C01785=1051.744,309.369,-107.707,172.758,38.228,157.251
C01786=1051.737,309.122,-107.673,172.754,38.225,157.251
C01787=1051.730,308.873,-107.640,172.750,38.221,157.250
C01788=1051.724,308.627,-107.607,172.747,38.218,157.249
C01789=1051.717,308.378,-107.574,172.743,38.214,157.248
C01790=1051.710,308.131,-107.541,172.739,38.211,157.247
C01791=1051.703,307.883,-107.507,172.737,38.207,157.246
C01792=1051.697,307.635,-107.474,172.733,38.203,157.245
C01793=1051.691,307.388,-107.441,172.729,38.200,157.245
C01794=1051.683,307.140,-107.409,172.725,38.197,157.244
C01795=1051.676,306.893,-107.375,172.722,38.193,157.243
C01796=1051.669,306.644,-107.342,172.719,38.189,157.242
C01797=1051.663,306.397,-107.310,172.715,38.186,157.241
C01798=1051.657,306.149,-107.277,172.712,38.183,157.240
C01799=1051.650,305.902,-107.243,172.708,38.179,157.239
C01800=1051.643,305.654,-107.210,172.704,38.175,157.239
C01801=1051.637,305.406,-107.178,172.701,38.172,157.238
C01802=1051.629,305.158,-107.145,172.698,38.168,157.237
C01803=1051.623,304.877,-107.108,172.694,38.164,157.236
C01804=1051.615,304.595,-107.070,172.690,38.160,157.235
C01805=1051.607,304.314,-107.033,172.685,38.156,157.234
C01806=1051.600,304.032,-106.996,172.682,38.152,157.233
C01807=1051.593,303.784,-106.963,172.679,38.149,157.232
C01808=1051.586,303.536,-106.930,172.675,38.145,157.231
C01809=1051.580,303.289,-106.898,172.671,38.141,157.230
C01810=1051.574,303.041,-106.865,172.668,38.138,157.230
C01811=1051.567,302.793,-106.832,172.665,38.135,157.229
C01812=1051.561,302.545,-106.799,172.661,38.131,157.228
C01813=1051.554,302.298,-106.766,172.658,38.128,157.227
C01814=1051.547,302.050,-106.734,172.655,38.124,157.226
C01815=1051.541,301.803,-106.701,172.651,38.120,157.225
C01816=1051.534,301.555,-106.668,172.648,38.117,157.225
C01817=1051.528,301.307,-106.636,172.644,38.114,157.224
C01818=1051.521,301.059,-106.603,172.641,38.110,157.223
C01819=1051.515,300.812,-106.570,172.638,38.106,157.222
C01820=1051.508,300.565,-106.538,172.634,38.103,157.221
C01821=1051.501,300.316,-106.505,172.631,38.099,157.220
C01822=1051.495,300.069,-106.472,172.628,38.096,157.220
C01823=1051.489,299.820,-106.440,172.624,38.093,157.219
C01824=1051.483,299.573,-106.407,172.621,38.089,157.218
C01825=1051.476,299.326,-106.375,172.618,38.085,157.217
C01826=1051.469,299.078,-106.342,172.614,38.082,157.216
C01827=1051.463,298.830,-106.310,172.611,38.078,157.215
C01828=1051.457,298.582,-106.278,172.608,38.075,157.215
C01829=1051.450,298.334,-106.245,172.604,38.072,157.214
C01830=1051.443,298.087,-106.212,172.601,38.068,157.213
C01831=1051.437,297.838,-106.180,172.598,38.065,157.212
C01832=1051.431,297.591,-106.148,172.595,38.061,157.211
C01833=1051.425,297.343,-106.115,172.591,38.057,157.210
C01834=1051.419,297.095,-106.083,172.587,38.054,157.210
C01835=1051.412,296.848,-106.051,172.585,38.051,157.209
C01836=1051.405,296.600,-106.018,172.581,38.047,157.208
C01837=1051.399,296.352,-105.986,172.578,38.044,157.207
C01838=1051.392,296.105,-105.954,172.575,38.040,157.206
C01839=1051.386,295.856,-105.922,172.571,38.037,157.205
C01840=1051.379,295.609,-105.890,172.569,38.033,157.205
C01841=1051.373,295.361,-105.858,172.565,38.030,157.204
C01842=1051.366,295.114,-105.825,172.561,38.027,157.203
C01843=1051.360,294.865,-105.793,172.559,38.023,157.202
C01844=1051.353,294.617,-105.761,172.555,38.020,157.201
C01845=1051.347,294.369,-105.729,172.552,38.016,157.201
C01846=1051.340,294.122,-105.697,172.549,38.013,157.200
C01847=1051.334,293.874,-105.665,172.545,38.010,157.199
C01848=1051.327,293.626,-105.633,172.542,38.006,157.198
C01849=1051.320,293.379,-105.601,172.539,38.003,157.197
C01850=1051.314,293.130,-105.569,172.536,37.999,157.197
C01851=1051.307,292.882,-105.538,172.533,37.996,157.196
C01852=1051.300,292.635,-105.506,172.529,37.993,157.195
C01853=1051.294,292.387,-105.474,172.526,37.990,157.194
C01854=1051.287,292.139,-105.442,172.523,37.986,157.193
C01855=1051.281,291.891,-105.410,172.520,37.983,157.193
C01856=1051.274,291.644,-105.378,172.516,37.979,157.192
C01857=1051.268,291.396,-105.346,172.513,37.976,157.191
C01858=1051.262,291.147,-105.314,172.510,37.972,157.190
C01859=1051.255,290.882,-105.280,172.506,37.969,157.189
C01860=1051.247,290.617,-105.247,172.503,37.966,157.189
C01861=1051.240,290.351,-105.213,172.500,37.962,157.188
C01862=1051.233,290.085,-105.179,172.496,37.958,157.187
C01863=1051.226,289.838,-105.147,172.493,37.955,157.186
C01864=1051.220,289.589,-105.115,172.490,37.952,157.185
C01865=1051.213,289.341,-105.083,172.487,37.949,157.185
C01866=1051.207,289.094,-105.052,172.484,37.945,157.184
C01867=1051.201,288.846,-105.020,172.480,37.942,157.183
C01868=1051.195,288.598,-104.989,172.478,37.938,157.182
C01869=1051.188,288.350,-104.957,172.474,37.935,157.181
C01870=1051.181,288.102,-104.926,172.471,37.932,157.181
C01871=1051.175,287.854,-104.894,172.468,37.929,157.180
C01872=1051.168,287.606,-104.862,172.465,37.925,157.179
C01873=1051.162,287.358,-104.831,172.462,37.922,157.178
C01874=1051.155,287.110,-104.800,172.459,37.919,157.178
C01875=1051.148,286.863,-104.768,172.455,37.915,157.177
C01876=1051.142,286.615,-104.737,172.453,37.912,157.176
C01877=1051.135,286.367,-104.706,172.449,37.909,157.175
C01878=1051.129,286.120,-104.674,172.447,37.906,157.175
C01879=1051.122,285.871,-104.644,172.443,37.902,157.174
C01880=1051.116,285.623,-104.612,172.440,37.899,157.173
C01881=1051.109,285.375,-104.581,172.437,37.896,157.172
C01882=1051.102,285.127,-104.549,172.434,37.892,157.171
C01883=1051.095,284.879,-104.518,172.431,37.889,157.171
C01884=1051.089,284.632,-104.486,172.428,37.886,157.170
C01885=1051.083,284.384,-104.456,172.424,37.883,157.169
C01886=1051.076,284.136,-104.425,172.422,37.879,157.168
C01887=1051.069,283.888,-104.393,172.418,37.876,157.168
C01888=1051.063,283.640,-104.361,172.416,37.873,157.167
C01889=1051.057,283.391,-104.330,172.412,37.870,157.166
C01890=1051.051,283.144,-104.299,172.409,37.866,157.165
C01891=1051.044,282.896,-104.268,172.406,37.863,157.165
C01892=1051.038,282.648,-104.237,172.403,37.860,157.164
C01893=1051.031,282.400,-104.206,172.401,37.856,157.163
C01894=1051.024,282.152,-104.174,172.397,37.853,157.162
C01895=1051.018,281.904,-104.144,172.394,37.850,157.162
C01896=1051.012,281.656,-104.113,172.391,37.847,157.161
C01897=1051.005,281.408,-104.081,172.388,37.844,157.160
C01898=1050.999,281.160,-104.050,172.385,37.840,157.159
C01899=1050.992,280.912,-104.019,172.382,37.837,157.159
C01900=1050.986,280.664,-103.989,172.379,37.833,157.158
C01901=1050.979,280.416,-103.957,172.376,37.830,157.157
C01902=1050.973,280.169,-103.926,172.373,37.827,157.156
C01903=1050.967,279.920,-103.895,172.370,37.824,157.155
C01904=1050.960,279.672,-103.864,172.367,37.821,157.155
C01905=1050.954,279.424,-103.834,172.365,37.817,157.154
C01906=1050.947,279.177,-103.803,172.361,37.814,157.153
C01907=1050.940,278.928,-103.772,172.358,37.811,157.153
C01908=1050.934,278.680,-103.741,172.355,37.807,157.152
C01909=1050.928,278.433,-103.710,172.352,37.805,157.151
C01910=1050.921,278.184,-103.680,172.349,37.801,157.150
C01911=1050.914,277.937,-103.649,172.346,37.798,157.150
C01912=1050.908,277.689,-103.618,172.344,37.795,157.149
C01913=1050.902,277.440,-103.588,172.340,37.791,157.148
C01914=1050.895,277.192,-103.556,172.337,37.788,157.147
C01915=1050.889,276.938,-103.525,172.335,37.785,157.147
C01916=1050.882,276.684,-103.493,172.331,37.782,157.146
C01917=1050.875,276.430,-103.462,172.329,37.779,157.145
C01918=1050.868,276.175,-103.431,172.325,37.775,157.144
C01919=1050.862,275.927,-103.400,172.322,37.772,157.144
C01920=1050.855,275.679,-103.370,172.320,37.769,157.143
C01921=1050.849,275.432,-103.339,172.316,37.765,157.142
C01922=1050.843,275.184,-103.308,172.314,37.762,157.141
C01923=1050.836,274.935,-103.278,172.310,37.759,157.141
C01924=1050.830,274.688,-103.248,172.308,37.756,157.140
C01925=1050.823,274.439,-103.217,172.305,37.753,157.139
C01926=1050.816,274.191,-103.186,172.302,37.750,157.138
C01927=1050.810,273.944,-103.156,172.299,37.746,157.138
C01928=1050.803,273.695,-103.125,172.296,37.743,157.137
C01929=1050.798,273.447,-103.095,172.293,37.740,157.136
C01930=1050.791,273.199,-103.065,172.290,37.737,157.135
C01931=1050.785,272.951,-103.034,172.288,37.734,157.135
C01932=1050.778,272.703,-103.004,172.284,37.730,157.134
C01933=1050.771,272.454,-102.974,172.282,37.727,157.133
C01934=1050.765,272.207,-102.943,172.279,37.724,157.133
C01935=1050.759,271.959,-102.912,172.276,37.721,157.132
C01936=1050.752,271.711,-102.882,172.273,37.717,157.131
C01937=1050.746,271.463,-102.851,172.270,37.715,157.130
C01938=1050.739,271.215,-102.822,172.268,37.711,157.130
C01939=1050.733,270.967,-102.791,172.264,37.708,157.129
C01940=1050.726,270.719,-102.762,172.262,37.705,157.128
C01941=1050.720,270.470,-102.731,172.259,37.702,157.128
C01942=1050.713,270.222,-102.701,172.256,37.698,157.127
C01943=1050.707,269.974,-102.671,172.253,37.695,157.126
C01944=1050.700,269.726,-102.640,172.250,37.692,157.125
C01945=1050.694,269.478,-102.610,172.248,37.689,157.125
C01946=1050.687,269.230,-102.580,172.244,37.686,157.124
C01947=1050.681,268.982,-102.550,172.242,37.683,157.123
C01948=1050.674,268.734,-102.520,172.239,37.680,157.123
C01949=1050.668,268.486,-102.489,172.237,37.676,157.122
C01950=1050.662,268.238,-102.460,172.233,37.673,157.121
C01951=1050.655,267.989,-102.429,172.231,37.670,157.120
C01952=1050.649,267.742,-102.400,172.228,37.667,157.120
C01953=1050.642,267.493,-102.370,172.225,37.664,157.119
C01954=1050.636,267.245,-102.340,172.222,37.661,157.118
C01955=1050.629,266.997,-102.310,172.220,37.658,157.117
C01956=1050.622,266.749,-102.280,172.217,37.654,157.117
C01957=1050.616,266.501,-102.249,172.213,37.651,157.116
C01958=1050.610,266.253,-102.220,172.211,37.648,157.115
C01959=1050.603,266.004,-102.190,172.208,37.645,157.115
C01960=1050.597,265.757,-102.160,172.206,37.642,157.114
C01961=1050.590,265.508,-102.130,172.203,37.639,157.113
C01962=1050.584,265.260,-102.100,172.200,37.636,157.112
C01963=1050.578,265.012,-102.070,172.197,37.632,157.112
C01964=1050.571,264.764,-102.041,172.195,37.629,157.111
C01965=1050.565,264.516,-102.011,172.192,37.626,157.110
C01966=1050.558,264.268,-101.980,172.189,37.623,157.110
C01967=1050.552,264.019,-101.951,172.186,37.619,157.109
C01968=1050.546,263.772,-101.921,172.183,37.617,157.108
C01969=1050.539,263.523,-101.892,172.181,37.614,157.108
C01970=1050.532,263.275,-101.862,172.178,37.610,157.107
C01971=1050.526,263.025,-101.832,172.175,37.607,157.106
C01972=1050.520,262.776,-101.802,172.172,37.604,157.105
C01973=1050.513,262.526,-101.772,172.170,37.601,157.105
C01974=1050.507,262.275,-101.742,172.167,37.598,157.104
C01975=1050.500,262.026,-101.713,172.165,37.594,157.103
C01976=1050.493,261.779,-101.683,172.161,37.592,157.103
C01977=1050.487,261.531,-101.654,172.159,37.589,157.102
C01978=1050.479,261.283,-101.624,172.156,37.586,157.101
C01979=1050.473,261.035,-101.595,172.154,37.582,157.100
C01980=1050.466,260.786,-101.566,172.150,37.579,157.100
C01981=1050.459,260.538,-101.536,172.148,37.576,157.099
C01982=1050.453,260.290,-101.507,172.145,37.573,157.098
C01983=1050.446,260.041,-101.478,172.143,37.570,157.098
C01984=1050.440,259.794,-101.448,172.140,37.567,157.097
C01985=1050.434,259.546,-101.419,172.138,37.564,157.096
C01986=1050.427,259.297,-101.390,172.134,37.561,157.096
C01987=1050.420,259.049,-101.361,172.132,37.558,157.095
C01988=1050.414,258.801,-101.331,172.129,37.555,157.094
C01989=1050.407,258.553,-101.301,172.127,37.552,157.094
C01990=1050.401,258.304,-101.272,172.124,37.548,157.093
C01991=1050.395,258.056,-101.243,172.122,37.546,157.092
C01992=1050.387,257.808,-101.213,172.118,37.543,157.092
C01993=1050.381,257.560,-101.184,172.115,37.539,157.091
C01994=1050.375,257.312,-101.155,172.113,37.536,157.090
C01995=1050.368,257.063,-101.126,172.111,37.533,157.089
C01996=1050.362,256.815,-101.097,172.108,37.530,157.089
C01997=1050.356,256.567,-101.068,172.105,37.527,157.088
C01998=1050.349,256.319,-101.038,172.103,37.524,157.087
C01999=1050.342,256.070,-101.008,172.099,37.521,157.087
C02000=1050.336,255.822,-100.979,172.097,37.518,157.086
C02001=1050.329,255.574,-100.951,172.094,37.515,157.085
C02002=1050.323,255.326,-100.922,172.092,37.512,157.085
C02003=1050.316,255.077,-100.893,172.089,37.508,157.084
C02004=1050.310,254.829,-100.864,172.087,37.505,157.083
C02005=1050.303,254.581,-100.834,172.084,37.502,157.083
C02006=1050.297,254.333,-100.805,172.082,37.499,157.082
C02007=1050.291,254.085,-100.776,172.079,37.496,157.081
C02008=1050.284,253.836,-100.747,172.077,37.493,157.080
C02009=1050.278,253.588,-100.718,172.073,37.490,157.080
C02010=1050.271,253.340,-100.689,172.071,37.487,157.079
C02011=1050.265,253.092,-100.660,172.068,37.484,157.078
C02012=1050.258,252.844,-100.631,172.066,37.480,157.078
C02013=1050.251,252.595,-100.602,172.063,37.477,157.077
C02014=1050.245,252.347,-100.573,172.061,37.474,157.076
C02015=1050.239,252.099,-100.544,172.058,37.471,157.076
C02016=1050.233,251.851,-100.515,172.056,37.468,157.075
C02017=1050.226,251.602,-100.486,172.053,37.465,157.074
C02018=1050.220,251.354,-100.457,172.051,37.461,157.073
C02019=1050.214,251.106,-100.428,172.048,37.458,157.073
C02020=1050.208,250.858,-100.399,172.046,37.456,157.072
C02021=1050.201,250.609,-100.370,172.043,37.452,157.071
C02022=1050.194,250.361,-100.342,172.041,37.449,157.071
C02023=1050.188,250.113,-100.313,172.038,37.446,157.070
C02024=1050.182,249.865,-100.284,172.036,37.443,157.069
C02025=1050.175,249.616,-100.254,172.033,37.440,157.069
C02026=1050.169,249.368,-100.225,172.031,37.437,157.068
C02027=1050.162,249.116,-100.196,172.028,37.433,157.067
C02028=1050.156,248.865,-100.167,172.026,37.430,157.067
C02029=1050.150,248.613,-100.138,172.022,37.427,157.066
C02030=1050.144,248.362,-100.109,172.020,37.424,157.065
C02031=1050.138,248.114,-100.081,172.017,37.420,157.064
C02032=1050.131,247.865,-100.052,172.015,37.417,157.064
C02033=1050.125,247.617,-100.023,172.012,37.415,157.063
C02034=1050.119,247.369,-99.993,172.010,37.411,157.062
C02035=1050.112,247.121,-99.966,172.007,37.408,157.062
C02036=1050.106,246.873,-99.937,172.005,37.405,157.061
C02037=1050.100,246.625,-99.908,172.003,37.402,157.060
C02038=1050.094,246.376,-99.879,172.001,37.399,157.060
C02039=1050.087,246.128,-99.850,171.998,37.395,157.059
C02040=1050.081,245.879,-99.821,171.996,37.392,157.058
C02041=1050.075,245.631,-99.794,171.993,37.389,157.057
C02042=1050.068,245.382,-99.764,171.991,37.386,157.057
C02043=1050.062,245.133,-99.736,171.988,37.383,157.056
C02044=1050.055,244.886,-99.707,171.986,37.380,157.055
C02045=1050.049,244.637,-99.679,171.983,37.376,157.055
C02046=1050.042,244.389,-99.651,171.981,37.373,157.054
C02047=1050.036,244.141,-99.622,171.978,37.370,157.053
C02048=1050.030,243.892,-99.593,171.976,37.367,157.053
C02049=1050.023,243.644,-99.565,171.973,37.364,157.052
C02050=1050.017,243.396,-99.536,171.971,37.361,157.051
C02051=1050.011,243.148,-99.509,171.968,37.358,157.051
C02052=1050.004,242.900,-99.480,171.966,37.355,157.050
C02053=1049.998,242.651,-99.452,171.963,37.352,157.049
C02054=1049.991,242.403,-99.423,171.961,37.349,157.049
C02055=1049.986,242.154,-99.395,171.958,37.345,157.048
C02056=1049.979,241.907,-99.367,171.956,37.342,157.047
C02057=1049.973,241.658,-99.338,171.953,37.339,157.047
C02058=1049.966,241.409,-99.310,171.951,37.336,157.046
C02059=1049.960,241.161,-99.281,171.948,37.333,157.045
C02060=1049.953,240.913,-99.254,171.946,37.330,157.044
C02061=1049.946,240.664,-99.226,171.943,37.327,157.044
C02062=1049.940,240.416,-99.197,171.942,37.323,157.043
C02063=1049.933,240.168,-99.169,171.939,37.320,157.042
C02064=1049.927,239.919,-99.141,171.937,37.317,157.042
C02065=1049.921,239.671,-99.113,171.934,37.314,157.041
C02066=1049.914,239.423,-99.085,171.932,37.311,157.040
C02067=1049.908,239.174,-99.056,171.929,37.308,157.040
C02068=1049.901,238.926,-99.029,171.927,37.305,157.039
C02069=1049.894,238.677,-99.001,171.924,37.302,157.038
C02070=1049.888,238.429,-98.972,171.922,37.299,157.038
C02071=1049.882,238.181,-98.944,171.919,37.296,157.037
C02072=1049.875,237.933,-98.917,171.917,37.293,157.036
C02073=1049.869,237.684,-98.888,171.915,37.290,157.036
C02074=1049.863,237.436,-98.861,171.913,37.286,157.035
C02075=1049.856,237.187,-98.833,171.911,37.283,157.034
C02076=1049.849,236.939,-98.805,171.908,37.280,157.034
C02077=1049.843,236.691,-98.776,171.906,37.277,157.033
C02078=1049.837,236.442,-98.748,171.903,37.274,157.032
C02079=1049.830,236.194,-98.721,171.901,37.271,157.032
C02080=1049.824,235.946,-98.693,171.898,37.268,157.031
C02081=1049.818,235.697,-98.665,171.896,37.265,157.030
C02082=1049.811,235.449,-98.637,171.893,37.261,157.030
C02083=1049.805,235.191,-98.608,171.892,37.258,157.029
C02084=1049.797,234.934,-98.579,171.889,37.255,157.028
C02085=1049.792,234.677,-98.550,171.887,37.252,157.027
C02086=1049.784,234.419,-98.522,171.884,37.248,157.027
C02087=1049.778,234.171,-98.493,171.882,37.245,157.026
C02088=1049.772,233.922,-98.466,171.879,37.242,157.025
C02089=1049.765,233.674,-98.438,171.877,37.239,157.025
C02090=1049.759,233.426,-98.411,171.874,37.236,157.024
C02091=1049.753,233.177,-98.382,171.873,37.233,157.023
C02092=1049.746,232.929,-98.355,171.870,37.230,157.023
C02093=1049.740,232.680,-98.327,171.868,37.226,157.022
C02094=1049.733,232.432,-98.299,171.865,37.224,157.021
C02095=1049.727,232.184,-98.272,171.863,37.221,157.021
C02096=1049.721,231.935,-98.244,171.860,37.217,157.020
C02097=1049.715,231.686,-98.216,171.859,37.214,157.019
C02098=1049.708,231.438,-98.189,171.857,37.211,157.019
C02099=1049.702,231.190,-98.161,171.854,37.208,157.018
C02100=1049.695,230.942,-98.134,171.852,37.205,157.017
C02101=1049.689,230.693,-98.106,171.849,37.202,157.017
C02102=1049.682,230.445,-98.078,171.847,37.199,157.016
C02103=1049.676,230.197,-98.051,171.845,37.195,157.015
C02104=1049.669,229.948,-98.024,171.843,37.192,157.015
C02105=1049.663,229.699,-97.995,171.840,37.189,157.014
C02106=1049.657,229.451,-97.968,171.838,37.186,157.013
C02107=1049.651,229.203,-97.940,171.835,37.183,157.013
C02108=1049.644,228.954,-97.913,171.834,37.180,157.012
C02109=1049.638,228.706,-97.886,171.831,37.177,157.011
C02110=1049.631,228.457,-97.858,171.829,37.173,157.010
C02111=1049.625,228.209,-97.831,171.826,37.170,157.010
C02112=1049.618,227.961,-97.804,171.824,37.167,157.009
C02113=1049.611,227.712,-97.776,171.823,37.164,157.009
C02114=1049.605,227.463,-97.749,171.820,37.161,157.008
C02115=1049.599,227.216,-97.722,171.818,37.158,157.007
C02116=1049.592,226.967,-97.694,171.815,37.155,157.007
C02117=1049.586,226.718,-97.667,171.814,37.152,157.006
C02118=1049.579,226.470,-97.639,171.811,37.148,157.005
C02119=1049.573,226.221,-97.613,171.809,37.145,157.004
C02120=1049.566,225.973,-97.585,171.806,37.142,157.004
C02121=1049.559,225.725,-97.558,171.804,37.139,157.003
C02122=1049.553,225.476,-97.531,171.802,37.136,157.002
C02123=1049.547,225.228,-97.504,171.800,37.133,157.002
C02124=1049.540,224.979,-97.477,171.797,37.130,157.001
C02125=1049.534,224.731,-97.449,171.795,37.126,157.000
C02126=1049.528,224.482,-97.422,171.794,37.123,157.000
C02127=1049.521,224.234,-97.394,171.791,37.120,156.999
C02128=1049.515,223.985,-97.368,171.789,37.117,156.999
C02129=1049.508,223.737,-97.341,171.786,37.114,156.998
C02130=1049.502,223.489,-97.314,171.785,37.111,156.997
C02131=1049.495,223.240,-97.286,171.782,37.108,156.996
C02132=1049.489,222.991,-97.259,171.780,37.104,156.996
C02133=1049.483,222.744,-97.232,171.778,37.101,156.995
C02134=1049.477,222.494,-97.205,171.776,37.098,156.994
C02135=1049.470,222.246,-97.177,171.773,37.095,156.994
C02136=1049.463,221.998,-97.151,171.771,37.092,156.993
C02137=1049.457,221.750,-97.123,171.770,37.089,156.992
C02138=1049.451,221.501,-97.097,171.767,37.085,156.992
C02139=1049.445,221.236,-97.068,171.765,37.082,156.991
C02140=1049.437,220.971,-97.039,171.762,37.079,156.990
C02141=1049.430,220.706,-97.011,171.761,37.075,156.990
C02142=1049.424,220.441,-96.981,171.758,37.072,156.989
C02143=1049.417,220.192,-96.954,171.756,37.069,156.988
C02144=1049.411,219.944,-96.928,171.753,37.066,156.987
C02145=1049.404,219.696,-96.901,171.752,37.063,156.987
C02146=1049.398,219.447,-96.874,171.749,37.059,156.986
C02147=1049.391,219.199,-96.847,171.747,37.056,156.985
C02148=1049.385,218.950,-96.820,171.744,37.053,156.985
C02149=1049.378,218.702,-96.794,171.743,37.050,156.984
C02150=1049.371,218.453,-96.767,171.740,37.047,156.983
C02151=1049.365,218.205,-96.741,171.738,37.044,156.983
C02152=1049.359,217.956,-96.714,171.737,37.041,156.982
C02153=1049.352,217.708,-96.686,171.734,37.038,156.982
C02154=1049.345,217.460,-96.660,171.732,37.034,156.981
C02155=1049.339,217.211,-96.633,171.730,37.031,156.980
C02156=1049.333,216.962,-96.607,171.728,37.028,156.979
C02157=1049.326,216.713,-96.580,171.725,37.024,156.979
C02158=1049.320,216.465,-96.553,171.724,37.021,156.978
C02159=1049.313,216.217,-96.526,171.721,37.018,156.977
C02160=1049.307,215.969,-96.499,171.719,37.015,156.977
C02161=1049.300,215.720,-96.473,171.717,37.012,156.976
C02162=1049.294,215.471,-96.446,171.715,37.009,156.975
C02163=1049.287,215.223,-96.420,171.713,37.005,156.975
C02164=1049.281,214.974,-96.393,171.711,37.002,156.974
C02165=1049.275,214.725,-96.366,171.709,36.999,156.973
C02166=1049.269,214.477,-96.340,171.707,36.996,156.973
C02167=1049.262,214.228,-96.313,171.705,36.993,156.972
C02168=1049.256,213.980,-96.287,171.702,36.989,156.971
C02169=1049.250,213.732,-96.260,171.701,36.986,156.971
C02170=1049.243,213.483,-96.234,171.698,36.983,156.970
C02171=1049.237,213.235,-96.207,171.696,36.980,156.969
C02172=1049.230,212.986,-96.181,171.695,36.977,156.969
C02173=1049.224,212.738,-96.154,171.692,36.974,156.968
C02174=1049.217,212.489,-96.128,171.691,36.970,156.967
C02175=1049.211,212.240,-96.101,171.688,36.967,156.967
C02176=1049.204,211.992,-96.075,171.686,36.964,156.966
C02177=1049.198,211.743,-96.048,171.684,36.961,156.965
C02178=1049.192,211.495,-96.022,171.682,36.958,156.965
C02179=1049.185,211.246,-95.995,171.680,36.954,156.964
C02180=1049.179,210.998,-95.969,171.678,36.951,156.963
C02181=1049.172,210.749,-95.943,171.676,36.948,156.963
C02182=1049.166,210.501,-95.916,171.674,36.944,156.962
C02183=1049.159,210.252,-95.890,171.672,36.941,156.961
C02184=1049.153,210.004,-95.863,171.670,36.938,156.960
C02185=1049.147,209.755,-95.838,171.668,36.935,156.960
C02186=1049.140,209.507,-95.811,171.665,36.932,156.959
C02187=1049.134,209.258,-95.784,171.664,36.928,156.958
C02188=1049.127,209.009,-95.758,171.661,36.925,156.958
C02189=1049.120,208.761,-95.732,171.660,36.922,156.957
C02190=1049.114,208.513,-95.707,171.657,36.919,156.956
C02191=1049.108,208.264,-95.680,171.656,36.916,156.956
C02192=1049.101,208.016,-95.654,171.654,36.912,156.955
C02193=1049.095,207.768,-95.628,171.651,36.909,156.954
C02194=1049.088,207.518,-95.601,171.650,36.906,156.954
C02195=1049.082,207.258,-95.574,171.647,36.903,156.953
C02196=1049.075,207.000,-95.547,171.646,36.899,156.952
C02197=1049.068,206.740,-95.519,171.643,36.896,156.952
C02198=1049.061,206.481,-95.492,171.641,36.892,156.951
C02199=1049.035,205.428,-95.386,171.404,36.795,156.930
C02200=1049.029,205.180,-95.361,171.402,36.792,156.929
C02201=1049.023,204.932,-95.336,171.400,36.790,156.929
C02202=1049.017,204.683,-95.311,171.396,36.788,156.928
C02203=1049.011,204.434,-95.286,171.394,36.785,156.928
C02204=1049.005,204.185,-95.261,171.392,36.783,156.927
C02205=1048.999,203.936,-95.235,171.388,36.780,156.927
C02206=1048.993,203.688,-95.211,171.386,36.778,156.926
C02207=1048.987,203.439,-95.186,171.384,36.776,156.926
C02208=1048.981,203.190,-95.161,171.382,36.773,156.925
C02209=1048.974,202.942,-95.136,171.378,36.771,156.925
C02210=1048.969,202.694,-95.112,171.376,36.768,156.924
C02211=1048.963,202.445,-95.086,171.374,36.766,156.924
C02212=1048.957,202.196,-95.062,171.370,36.763,156.923
C02213=1048.951,201.947,-95.036,171.368,36.761,156.923
C02214=1048.945,201.699,-95.011,171.366,36.759,156.923
C02215=1048.939,201.450,-94.987,171.363,36.756,156.922
C02216=1048.932,201.201,-94.962,171.360,36.754,156.922
C02217=1048.926,200.952,-94.937,171.358,36.752,156.921
C02218=1048.921,200.704,-94.912,171.355,36.750,156.921
C02219=1048.914,200.455,-94.888,171.352,36.747,156.920
C02220=1048.908,200.206,-94.863,171.350,36.745,156.920
C02221=1048.902,199.957,-94.838,171.348,36.742,156.919
C02222=1048.895,199.709,-94.814,171.345,36.741,156.919
C02223=1048.890,199.460,-94.789,171.342,36.738,156.918
C02224=1048.883,199.211,-94.765,171.340,36.736,156.918
C02225=1048.877,198.963,-94.740,171.337,36.733,156.917
C02226=1048.871,198.714,-94.716,171.335,36.731,156.917
C02227=1048.865,198.466,-94.691,171.332,36.729,156.916
C02228=1048.859,198.216,-94.666,171.329,36.727,156.916
C02229=1048.852,197.968,-94.642,171.327,36.724,156.915
C02230=1048.847,197.719,-94.617,171.325,36.722,156.915
C02231=1048.840,197.470,-94.593,171.322,36.720,156.915
C02232=1048.834,197.222,-94.568,171.319,36.718,156.914
C02233=1048.828,196.973,-94.544,171.317,36.715,156.914
C02234=1048.822,196.724,-94.520,171.315,36.713,156.913
C02235=1048.816,196.475,-94.494,171.311,36.711,156.913
C02236=1048.809,196.227,-94.471,171.309,36.709,156.912
C02237=1048.804,195.978,-94.446,171.307,36.706,156.912
C02238=1048.797,195.729,-94.422,171.305,36.704,156.911
C02239=1048.791,195.481,-94.397,171.301,36.702,156.911
C02240=1048.785,195.232,-94.373,171.299,36.700,156.910
C02241=1048.779,194.983,-94.348,171.297,36.697,156.910
C02242=1048.774,194.734,-94.324,171.294,36.695,156.909
C02243=1048.767,194.486,-94.299,171.292,36.693,156.909
C02244=1048.761,194.237,-94.275,171.289,36.690,156.908
C02245=1048.755,193.988,-94.251,171.287,36.688,156.908
C02246=1048.749,193.739,-94.227,171.284,36.686,156.908
C02247=1048.742,193.491,-94.202,171.282,36.684,156.907
C02248=1048.736,193.242,-94.178,171.279,36.681,156.907
C02249=1048.730,192.994,-94.154,171.276,36.679,156.906
C02250=1048.725,192.744,-94.129,171.274,36.677,156.906
C02251=1048.719,192.496,-94.106,171.272,36.675,156.905
C02252=1048.713,192.247,-94.081,171.270,36.672,156.905
C02253=1048.706,191.998,-94.057,171.267,36.670,156.904
C02254=1048.700,191.750,-94.032,171.264,36.668,156.904
C02255=1048.694,191.501,-94.008,171.262,36.666,156.903
C02256=1048.688,191.252,-93.984,171.259,36.663,156.903
C02257=1048.683,191.003,-93.959,171.257,36.661,156.903
C02258=1048.676,190.755,-93.935,171.255,36.659,156.902
C02259=1048.671,190.505,-93.911,171.253,36.657,156.902
C02260=1048.664,190.221,-93.884,171.249,36.654,156.901
C02261=1048.657,189.937,-93.856,171.247,36.652,156.901
C02262=1048.650,189.652,-93.828,171.244,36.649,156.900
C02263=1048.643,189.369,-93.801,171.241,36.647,156.900
C02264=1048.637,189.119,-93.776,171.239,36.644,156.899
C02265=1048.631,188.871,-93.752,171.236,36.642,156.899
C02266=1048.625,188.622,-93.728,171.233,36.640,156.898
C02267=1048.619,188.374,-93.704,171.231,36.638,156.898
C02268=1048.613,188.124,-93.679,171.229,36.635,156.897
C02269=1048.607,187.876,-93.656,171.227,36.633,156.897
C02270=1048.602,187.627,-93.632,171.224,36.631,156.896
C02271=1048.596,187.378,-93.608,171.222,36.629,156.896
C02272=1048.590,187.129,-93.584,171.219,36.627,156.896
C02273=1048.584,186.880,-93.560,171.217,36.624,156.895
C02274=1048.578,186.632,-93.536,171.214,36.622,156.895
C02275=1048.572,186.383,-93.512,171.212,36.620,156.894
C02276=1048.566,186.134,-93.487,171.210,36.618,156.894
C02277=1048.560,185.886,-93.464,171.207,36.615,156.893
C02278=1048.554,185.637,-93.440,171.205,36.613,156.893
C02279=1048.548,185.388,-93.415,171.203,36.611,156.892
C02280=1048.543,185.139,-93.393,171.201,36.609,156.892
C02281=1048.537,184.890,-93.368,171.197,36.607,156.891
C02282=1048.531,184.642,-93.344,171.195,36.604,156.891
C02283=1048.525,184.393,-93.320,171.193,36.602,156.890
C02284=1048.519,184.144,-93.296,171.190,36.600,156.890
C02285=1048.514,183.895,-93.272,171.188,36.598,156.890
C02286=1048.507,183.646,-93.248,171.186,36.596,156.889
C02287=1048.501,183.398,-93.225,171.184,36.594,156.889
C02288=1048.494,183.148,-93.202,171.181,36.592,156.888
C02289=1048.488,182.900,-93.178,171.179,36.590,156.888
C02290=1048.481,182.651,-93.154,171.176,36.587,156.888
C02291=1048.476,182.402,-93.131,171.174,36.585,156.887
C02292=1048.469,182.153,-93.107,171.171,36.584,156.887
C02293=1048.463,181.904,-93.084,171.169,36.581,156.886
C02294=1048.457,181.656,-93.061,171.167,36.579,156.886
C02295=1048.451,181.407,-93.037,171.165,36.578,156.886
C02296=1048.445,181.158,-93.014,171.162,36.575,156.885
C02297=1048.438,180.909,-92.990,171.160,36.573,156.885
C02298=1048.432,180.660,-92.967,171.157,36.571,156.884
C02299=1048.426,180.411,-92.943,171.155,36.570,156.884
C02300=1048.420,180.163,-92.920,171.152,36.567,156.883
C02301=1048.414,179.914,-92.896,171.150,36.565,156.883
C02302=1048.408,179.665,-92.873,171.148,36.564,156.883
C02303=1048.401,179.417,-92.850,171.146,36.561,156.882
C02304=1048.395,179.168,-92.827,171.144,36.559,156.882
C02305=1048.389,178.919,-92.803,171.141,36.557,156.882
C02306=1048.383,178.670,-92.780,171.139,36.555,156.881
C02307=1048.376,178.421,-92.756,171.137,36.553,156.881
C02308=1048.371,178.172,-92.733,171.134,36.551,156.880
C02309=1048.364,177.924,-92.709,171.131,36.549,156.880
C02310=1048.358,177.674,-92.686,171.129,36.547,156.879
C02311=1048.352,177.426,-92.662,171.127,36.545,156.879
C02312=1048.346,177.177,-92.639,171.125,36.543,156.879
C02313=1048.340,176.927,-92.616,171.122,36.541,156.878
C02314=1048.333,176.679,-92.593,171.120,36.539,156.878
C02315=1048.328,176.431,-92.570,171.118,36.537,156.877
C02316=1048.321,176.182,-92.546,171.116,36.535,156.877
C02317=1048.315,175.933,-92.523,171.113,36.533,156.877
C02318=1048.309,175.684,-92.500,171.111,36.531,156.876
C02319=1048.303,175.436,-92.476,171.109,36.529,156.876
C02320=1048.297,175.186,-92.453,171.107,36.527,156.875
C02321=1048.291,174.937,-92.430,171.104,36.525,156.875
C02322=1048.285,174.689,-92.407,171.102,36.523,156.875
C02323=1048.279,174.440,-92.384,171.100,36.521,156.874
C02324=1048.272,174.155,-92.357,171.097,36.518,156.874
C02325=1048.264,173.870,-92.331,171.094,36.517,156.873
C02326=1048.258,173.585,-92.304,171.092,36.514,156.873
C02327=1048.251,173.300,-92.278,171.089,36.512,156.872
C02328=1048.245,173.052,-92.255,171.087,36.510,156.872
C02329=1048.239,172.803,-92.232,171.084,36.508,156.872
C02330=1048.233,172.554,-92.209,171.082,36.506,156.871
C02331=1048.227,172.305,-92.186,171.080,36.504,156.871
C02332=1048.221,172.056,-92.162,171.078,36.502,156.870
C02333=1048.215,171.807,-92.139,171.075,36.499,156.870
C02334=1048.209,171.558,-92.116,171.073,36.498,156.870
C02335=1048.203,171.310,-92.094,171.071,36.496,156.869
C02336=1048.197,171.060,-92.070,171.069,36.494,156.869
C02337=1048.190,170.812,-92.047,171.066,36.492,156.868
C02338=1048.185,170.563,-92.024,171.064,36.490,156.868
C02339=1048.179,170.314,-92.001,171.062,36.488,156.868
C02340=1048.173,170.065,-91.978,171.060,36.485,156.867
C02341=1048.167,169.817,-91.955,171.057,36.484,156.867
C02342=1048.161,169.568,-91.933,171.055,36.482,156.866
C02343=1048.155,169.318,-91.909,171.053,36.480,156.866
C02344=1048.149,169.069,-91.886,171.051,36.477,156.866
C02345=1048.143,168.821,-91.863,171.049,36.476,156.865
C02346=1048.137,168.572,-91.840,171.046,36.474,156.865
C02347=1048.131,168.324,-91.817,171.044,36.472,156.864
C02348=1048.125,168.075,-91.794,171.042,36.470,156.864
C02349=1048.119,167.826,-91.771,171.040,36.468,156.864
C02350=1048.114,167.577,-91.748,171.037,36.466,156.863
C02351=1048.108,167.328,-91.726,171.035,36.463,156.863
C02352=1048.102,167.078,-91.702,171.033,36.462,156.862
C02353=1048.095,166.830,-91.680,171.031,36.460,156.862
C02354=1048.089,166.581,-91.657,171.028,36.458,156.862
C02355=1048.084,166.332,-91.634,171.026,36.455,156.861
C02356=1048.078,166.083,-91.611,171.025,36.454,156.861
C02357=1048.072,165.834,-91.588,171.023,36.452,156.860
C02358=1048.066,165.586,-91.566,171.021,36.450,156.860
C02359=1048.060,165.337,-91.543,171.018,36.447,156.860
C02360=1048.054,165.088,-91.520,171.016,36.446,156.859
C02361=1048.048,164.839,-91.497,171.014,36.444,156.859
C02362=1048.043,164.590,-91.474,171.012,36.442,156.858
C02363=1048.036,164.341,-91.452,171.009,36.439,156.858
C02364=1048.031,164.093,-91.429,171.007,36.438,156.858
C02365=1048.025,163.843,-91.406,171.005,36.436,156.857
C02366=1048.019,163.594,-91.383,171.003,36.434,156.857
C02367=1048.013,163.346,-91.361,171.000,36.432,156.856
C02368=1048.007,163.097,-91.338,170.998,36.430,156.856
C02369=1048.001,162.848,-91.315,170.996,36.428,156.856
C02370=1047.996,162.599,-91.292,170.994,36.426,156.855
C02371=1047.990,162.350,-91.269,170.991,36.424,156.855
C02372=1047.984,162.101,-91.247,170.990,36.422,156.854
C02373=1047.978,161.852,-91.225,170.988,36.420,156.854
C02374=1047.972,161.603,-91.202,170.986,36.417,156.854
C02375=1047.967,161.354,-91.179,170.984,36.416,156.853
C02376=1047.960,161.106,-91.157,170.981,36.414,156.853
C02377=1047.954,160.857,-91.134,170.979,36.412,156.853
C02378=1047.949,160.607,-91.111,170.977,36.409,156.852
C02379=1047.943,160.359,-91.089,170.975,36.408,156.852
C02380=1047.937,160.110,-91.066,170.972,36.406,156.851
C02381=1047.931,159.860,-91.044,170.970,36.404,156.851
C02382=1047.925,159.612,-91.021,170.968,36.402,156.851
C02383=1047.918,159.363,-90.999,170.966,36.400,156.850
C02384=1047.912,159.114,-90.977,170.965,36.398,156.850
C02385=1047.907,158.865,-90.955,170.962,36.396,156.850
C02386=1047.900,158.616,-90.932,170.960,36.395,156.849
C02387=1047.895,158.367,-90.910,170.958,36.393,156.849
C02388=1047.888,158.082,-90.884,170.956,36.390,156.848
C02389=1047.881,157.796,-90.859,170.952,36.388,156.848
C02390=1047.873,157.511,-90.833,170.950,36.387,156.848
C02391=1047.867,157.226,-90.808,170.948,36.384,156.847
C02392=1047.860,156.978,-90.786,170.946,36.382,156.847
C02393=1047.855,156.728,-90.763,170.944,36.380,156.846
C02394=1047.848,156.480,-90.741,170.941,36.379,156.846
C02395=1047.843,156.230,-90.719,170.939,36.377,156.846
C02396=1047.836,155.981,-90.696,170.937,36.375,156.845
C02397=1047.830,155.732,-90.675,170.936,36.373,156.845
C02398=1047.824,155.483,-90.652,170.934,36.371,156.845
C02399=1047.818,155.234,-90.630,170.931,36.369,156.844
C02400=1047.812,154.986,-90.608,170.929,36.368,156.844
C02401=1047.807,154.737,-90.586,170.927,36.366,156.843
C02402=1047.800,154.488,-90.564,170.925,36.364,156.843
C02403=1047.794,154.239,-90.542,170.923,36.362,156.843
C02404=1047.788,153.990,-90.520,170.920,36.360,156.842
C02405=1047.782,153.741,-90.497,170.918,36.358,156.842
C02406=1047.776,153.492,-90.475,170.917,36.356,156.842
C02407=1047.770,153.243,-90.453,170.915,36.355,156.841
C02408=1047.764,152.994,-90.432,170.912,36.353,156.841
C02409=1047.758,152.745,-90.409,170.910,36.351,156.841
C02410=1047.752,152.496,-90.387,170.908,36.349,156.840
C02411=1047.745,152.247,-90.365,170.906,36.347,156.840
C02412=1047.740,151.999,-90.344,170.904,36.345,156.839
C02413=1047.734,151.749,-90.322,170.901,36.344,156.839
C02414=1047.728,151.501,-90.299,170.899,36.342,156.839
C02415=1047.722,151.251,-90.277,170.898,36.340,156.838
C02416=1047.715,151.002,-90.256,170.896,36.338,156.838
C02417=1047.709,150.754,-90.233,170.894,36.336,156.838
C02418=1047.704,150.504,-90.211,170.891,36.334,156.837
C02419=1047.698,150.256,-90.190,170.889,36.332,156.837
C02420=1047.692,150.007,-90.168,170.887,36.331,156.837
C02421=1047.685,149.758,-90.146,170.885,36.329,156.836
C02422=1047.679,149.509,-90.124,170.884,36.327,156.836
C02423=1047.673,149.260,-90.102,170.881,36.325,156.836
C02424=1047.667,149.010,-90.080,170.879,36.323,156.835
C02425=1047.662,148.762,-90.058,170.877,36.321,156.835
C02426=1047.656,148.513,-90.037,170.875,36.319,156.834
C02427=1047.649,148.264,-90.014,170.873,36.318,156.834
C02428=1047.643,148.015,-89.993,170.870,36.316,156.834
C02429=1047.637,147.766,-89.971,170.869,36.314,156.833
C02430=1047.631,147.517,-89.950,170.867,36.312,156.833
C02431=1047.625,147.268,-89.928,170.865,36.311,156.833
C02432=1047.619,147.019,-89.906,170.863,36.309,156.832
C02433=1047.612,146.770,-89.884,170.860,36.307,156.832
C02434=1047.606,146.521,-89.863,170.858,36.305,156.832
C02435=1047.600,146.272,-89.841,170.856,36.303,156.831
C02436=1047.595,146.023,-89.820,170.855,36.302,156.831
C02437=1047.588,145.774,-89.798,170.853,36.300,156.831
C02438=1047.582,145.525,-89.776,170.850,36.298,156.830
C02439=1047.576,145.276,-89.755,170.848,36.297,156.830
C02440=1047.570,145.026,-89.733,170.846,36.295,156.830
C02441=1047.564,144.779,-89.711,170.844,36.293,156.829
C02442=1047.558,144.529,-89.690,170.843,36.291,156.829
C02443=1047.552,144.280,-89.668,170.840,36.289,156.829
C02444=1047.546,144.031,-89.646,170.838,36.287,156.828
C02445=1047.539,143.782,-89.625,170.836,36.285,156.828
C02446=1047.534,143.533,-89.603,170.834,36.284,156.827
C02447=1047.528,143.284,-89.582,170.832,36.282,156.827
C02448=1047.522,143.035,-89.560,170.831,36.280,156.827
C02449=1047.515,142.786,-89.538,170.828,36.279,156.827
C02450=1047.510,142.537,-89.517,170.826,36.277,156.826
C02451=1047.503,142.288,-89.496,170.824,36.275,156.826
C02452=1047.497,142.003,-89.472,170.822,36.273,156.825
C02453=1047.489,141.717,-89.447,170.819,36.271,156.825
C02454=1047.483,141.432,-89.422,170.817,36.269,156.825
C02455=1047.475,141.146,-89.398,170.815,36.267,156.824
C02456=1047.470,140.897,-89.376,170.813,36.265,156.824
C02457=1047.464,140.648,-89.355,170.811,36.263,156.824
C02458=1047.457,140.399,-89.333,170.808,36.261,156.823
C02459=1047.452,140.150,-89.312,170.807,36.259,156.823
C02460=1047.446,139.901,-89.290,170.805,36.258,156.822
C02461=1047.439,139.652,-89.269,170.803,36.256,156.822
C02462=1047.433,139.403,-89.247,170.801,36.254,156.822
C02463=1047.427,139.154,-89.227,170.799,36.253,156.822
C02464=1047.421,138.905,-89.205,170.797,36.251,156.821
C02465=1047.415,138.655,-89.184,170.795,36.249,156.821
C02466=1047.409,138.407,-89.162,170.793,36.248,156.821
C02467=1047.403,138.158,-89.141,170.791,36.246,156.820
C02468=1047.396,137.909,-89.120,170.789,36.244,156.820
C02469=1047.391,137.660,-89.099,170.787,36.242,156.819
C02470=1047.385,137.410,-89.078,170.785,36.240,156.819
C02471=1047.378,137.161,-89.056,170.783,36.239,156.819
C02472=1047.373,136.913,-89.035,170.781,36.237,156.819
C02473=1047.366,136.664,-89.014,170.779,36.235,156.818
C02474=1047.360,136.414,-88.993,170.777,36.233,156.818
C02475=1047.354,136.166,-88.972,170.775,36.231,156.817
C02476=1047.348,135.917,-88.950,170.773,36.230,156.817
C02477=1047.342,135.667,-88.929,170.771,36.228,156.817
C02478=1047.336,135.419,-88.909,170.769,36.227,156.817
C02479=1047.330,135.169,-88.887,170.768,36.225,156.816
C02480=1047.324,134.920,-88.865,170.765,36.223,156.816
C02481=1047.318,134.671,-88.846,170.763,36.222,156.816
C02482=1047.311,134.422,-88.824,170.761,36.220,156.815
C02483=1047.306,134.174,-88.803,170.760,36.218,156.815
C02484=1047.299,133.924,-88.782,170.758,36.216,156.814
C02485=1047.293,133.675,-88.761,170.755,36.215,156.814
C02486=1047.288,133.426,-88.739,170.753,36.213,156.814
C02487=1047.281,133.177,-88.719,170.751,36.211,156.814
C02488=1047.275,132.928,-88.697,170.750,36.209,156.813
C02489=1047.269,132.679,-88.676,170.748,36.207,156.813
C02490=1047.263,132.430,-88.656,170.746,36.206,156.813
C02491=1047.257,132.181,-88.635,170.743,36.204,156.812
C02492=1047.251,131.931,-88.614,170.742,36.202,156.812
C02493=1047.245,131.683,-88.593,170.740,36.200,156.812
C02494=1047.239,131.434,-88.571,170.738,36.199,156.811
C02495=1047.233,131.184,-88.550,170.736,36.197,156.811
C02496=1047.227,130.936,-88.530,170.734,36.195,156.811
C02497=1047.220,130.686,-88.509,170.732,36.194,156.810
C02498=1047.214,130.437,-88.488,170.730,36.192,156.810
C02499=1047.208,130.188,-88.468,170.728,36.190,156.810
C02500=1047.201,129.939,-88.447,170.726,36.189,156.809
C02501=1047.196,129.690,-88.426,170.725,36.187,156.809
C02502=1047.189,129.441,-88.405,170.722,36.185,156.809
C02503=1047.183,129.192,-88.384,170.720,36.184,156.808
C02504=1047.177,128.943,-88.364,170.718,36.182,156.808
C02505=1047.170,128.694,-88.343,170.717,36.181,156.808
C02506=1047.165,128.445,-88.323,170.715,36.179,156.807
C02507=1047.158,128.196,-88.302,170.713,36.177,156.807
C02508=1047.152,127.947,-88.282,170.710,36.176,156.807
C02509=1047.146,127.698,-88.260,170.708,36.174,156.807
C02510=1047.139,127.448,-88.240,170.707,36.172,156.806
C02511=1047.133,127.200,-88.220,170.705,36.171,156.806
C02512=1047.127,126.950,-88.198,170.703,36.169,156.806
C02513=1047.121,126.702,-88.178,170.701,36.167,156.805
C02514=1047.115,126.452,-88.157,170.699,36.166,156.805
C02515=1047.109,126.204,-88.137,170.697,36.164,156.805
C02516=1047.101,125.917,-88.113,170.695,36.162,156.804
C02517=1047.094,125.632,-88.089,170.693,36.161,156.804
C02518=1047.087,125.346,-88.066,170.691,36.159,156.804
C02519=1047.080,125.061,-88.042,170.688,36.157,156.803
C02520=1047.075,124.811,-88.021,170.686,36.155,156.803
C02521=1047.068,124.563,-88.001,170.684,36.153,156.802
C02522=1047.062,124.313,-87.980,170.683,36.151,156.802
C02523=1047.056,124.064,-87.960,170.681,36.150,156.802
C02524=1047.050,123.815,-87.939,170.679,36.148,156.802
C02525=1047.044,123.566,-87.919,170.676,36.146,156.801
C02526=1047.038,123.316,-87.898,170.675,36.145,156.801
C02527=1047.032,123.068,-87.878,170.673,36.143,156.801
C02528=1047.025,122.819,-87.857,170.671,36.141,156.800
C02529=1047.019,122.570,-87.837,170.669,36.140,156.800
C02530=1047.013,122.320,-87.816,170.668,36.138,156.800
C02531=1047.007,122.071,-87.796,170.665,36.136,156.799
C02532=1047.000,121.822,-87.775,170.663,36.135,156.799
C02533=1046.995,121.573,-87.754,170.662,36.133,156.799
C02534=1046.988,121.324,-87.734,170.660,36.131,156.798
C02535=1046.982,121.075,-87.714,170.658,36.130,156.798
C02536=1046.977,120.826,-87.694,170.656,36.128,156.798
C02537=1046.970,120.577,-87.673,170.654,36.126,156.797
C02538=1046.964,120.328,-87.653,170.652,36.125,156.797
C02539=1046.958,120.078,-87.632,170.650,36.123,156.797
C02540=1046.952,119.829,-87.612,170.649,36.121,156.796
C02541=1046.946,119.581,-87.592,170.647,36.120,156.796
C02542=1046.940,119.331,-87.571,170.645,36.118,156.796
C02543=1046.934,119.082,-87.551,170.642,36.116,156.796
C02544=1046.927,118.833,-87.530,170.641,36.114,156.795
C02545=1046.921,118.584,-87.510,170.639,36.113,156.795
C02546=1046.916,118.335,-87.489,170.637,36.111,156.795
C02547=1046.910,118.086,-87.469,170.636,36.109,156.794
C02548=1046.904,117.837,-87.449,170.634,36.108,156.794
C02549=1046.898,117.588,-87.429,170.631,36.106,156.794
C02550=1046.892,117.338,-87.408,170.629,36.104,156.793
C02551=1046.886,117.089,-87.388,170.628,36.102,156.793
C02552=1046.880,116.841,-87.368,170.626,36.101,156.793
C02553=1046.874,116.591,-87.347,170.624,36.099,156.792
C02554=1046.868,116.342,-87.327,170.622,36.097,156.792
C02555=1046.862,116.093,-87.307,170.620,36.096,156.792
C02556=1046.856,115.844,-87.286,170.618,36.094,156.791
C02557=1046.850,115.595,-87.266,170.617,36.092,156.791
C02558=1046.844,115.346,-87.246,170.615,36.091,156.791
C02559=1046.837,115.097,-87.226,170.613,36.089,156.790
C02560=1046.832,114.848,-87.205,170.611,36.087,156.790
C02561=1046.826,114.599,-87.185,170.609,36.086,156.790
C02562=1046.819,114.349,-87.165,170.607,36.084,156.790
C02563=1046.813,114.101,-87.145,170.606,36.082,156.789
C02564=1046.808,113.851,-87.125,170.604,36.081,156.789
C02565=1046.802,113.601,-87.105,170.602,36.079,156.788
C02566=1046.796,113.352,-87.085,170.599,36.077,156.788
C02567=1046.790,113.104,-87.065,170.598,36.076,156.788
C02568=1046.783,112.854,-87.044,170.596,36.074,156.788
C02569=1046.777,112.605,-87.024,170.594,36.072,156.787
C02570=1046.771,112.356,-87.004,170.593,36.071,156.787
C02571=1046.765,112.107,-86.984,170.591,36.069,156.787
C02572=1046.759,111.858,-86.964,170.588,36.067,156.786
C02573=1046.753,111.609,-86.945,170.587,36.066,156.786
C02574=1046.747,111.360,-86.925,170.585,36.064,156.786
C02575=1046.740,111.110,-86.905,170.583,36.062,156.785
C02576=1046.734,110.862,-86.885,170.582,36.061,156.785
C02577=1046.728,110.613,-86.865,170.580,36.059,156.785
C02578=1046.722,110.363,-86.844,170.578,36.058,156.785
C02579=1046.716,110.114,-86.825,170.575,36.056,156.784
C02580=1046.709,109.828,-86.803,170.573,36.054,156.784
C02581=1046.702,109.542,-86.780,170.572,36.052,156.784
C02582=1046.695,109.256,-86.758,170.570,36.050,156.783
C02583=1046.688,108.971,-86.734,170.568,36.049,156.783
C02584=1046.681,108.721,-86.714,170.566,36.047,156.783
C02585=1046.674,108.472,-86.695,170.563,36.045,156.782
C02586=1046.668,108.224,-86.675,170.562,36.044,156.782
C02587=1046.663,107.974,-86.656,170.560,36.042,156.782
C02588=1046.656,107.725,-86.635,170.558,36.041,156.781
C02589=1046.650,107.476,-86.615,170.556,36.039,156.781
C02590=1046.644,107.227,-86.595,170.555,36.038,156.781
C02591=1046.638,106.977,-86.576,170.552,36.036,156.780
C02592=1046.631,106.728,-86.556,170.550,36.035,156.780
C02593=1046.625,106.480,-86.537,170.549,36.033,156.780
C02594=1046.620,106.230,-86.517,170.547,36.031,156.780
C02595=1046.614,105.981,-86.497,170.545,36.030,156.779
C02596=1046.607,105.731,-86.478,170.544,36.028,156.779
C02597=1046.601,105.482,-86.458,170.542,36.027,156.779
C02598=1046.595,105.234,-86.438,170.539,36.025,156.778
C02599=1046.589,104.984,-86.419,170.538,36.023,156.778
C02600=1046.582,104.735,-86.399,170.536,36.022,156.778
C02601=1046.576,104.486,-86.379,170.534,36.020,156.778
C02602=1046.571,104.237,-86.360,170.533,36.018,156.777
C02603=1046.565,103.988,-86.340,170.531,36.017,156.777
C02604=1046.558,103.739,-86.321,170.528,36.015,156.777
C02605=1046.552,103.489,-86.301,170.527,36.013,156.776
C02606=1046.546,103.240,-86.281,170.525,36.012,156.776
C02607=1046.540,102.991,-86.261,170.523,36.010,156.776
C02608=1046.534,102.742,-86.242,170.522,36.009,156.775
C02609=1046.528,102.493,-86.222,170.520,36.007,156.775
C02610=1046.521,102.244,-86.203,170.517,36.005,156.775
C02611=1046.515,101.994,-86.183,170.516,36.004,156.774
C02612=1046.509,101.745,-86.163,170.514,36.002,156.774
C02613=1046.503,101.496,-86.144,170.512,36.001,156.774
C02614=1046.497,101.247,-86.124,170.511,35.999,156.774
C02615=1046.491,100.998,-86.106,170.509,35.997,156.773
C02616=1046.485,100.749,-86.086,170.507,35.996,156.773
C02617=1046.479,100.500,-86.066,170.505,35.994,156.773
C02618=1046.473,100.250,-86.046,170.503,35.993,156.772
C02619=1046.466,100.001,-86.027,170.501,35.991,156.772
C02620=1046.461,99.752,-86.008,170.500,35.990,156.772
C02621=1046.454,99.503,-85.989,170.498,35.988,156.771
C02622=1046.448,99.254,-85.969,170.496,35.986,156.771
C02623=1046.441,99.004,-85.950,170.494,35.984,156.771
C02624=1046.435,98.755,-85.931,170.492,35.983,156.771
C02625=1046.429,98.506,-85.912,170.490,35.982,156.770
C02626=1046.423,98.257,-85.892,170.489,35.980,156.770
C02627=1046.417,98.008,-85.873,170.487,35.979,156.770
C02628=1046.411,97.759,-85.854,170.485,35.977,156.769
C02629=1046.405,97.510,-85.834,170.484,35.976,156.769
C02630=1046.398,97.260,-85.815,170.481,35.974,156.769
C02631=1046.392,97.010,-85.796,170.479,35.972,156.769
C02632=1046.385,96.762,-85.776,170.478,35.971,156.768
C02633=1046.380,96.512,-85.757,170.476,35.969,156.768
C02634=1046.373,96.263,-85.739,170.474,35.967,156.768
C02635=1046.367,96.015,-85.719,170.473,35.966,156.767
C02636=1046.361,95.765,-85.699,170.471,35.964,156.767
C02637=1046.355,95.516,-85.681,170.468,35.963,156.767
C02638=1046.349,95.267,-85.661,170.467,35.961,156.767
C02639=1046.342,95.017,-85.642,170.465,35.960,156.766
C02640=1046.336,94.768,-85.622,170.463,35.958,156.766
C02641=1046.330,94.519,-85.604,170.462,35.957,156.766
C02642=1046.324,94.269,-85.585,170.460,35.955,156.765
C02643=1046.317,94.021,-85.565,170.458,35.954,156.765
C02644=1046.310,93.735,-85.544,170.455,35.952,156.765
C02645=1046.304,93.449,-85.521,170.454,35.950,156.764
C02646=1046.297,93.163,-85.499,170.452,35.948,156.764
C02647=1046.290,92.877,-85.477,170.450,35.946,156.764
C02648=1046.283,92.628,-85.458,170.448,35.945,156.764
C02649=1046.278,92.379,-85.439,170.446,35.943,156.763
C02650=1046.271,92.130,-85.420,170.444,35.942,156.763
C02651=1046.265,91.880,-85.401,170.442,35.940,156.763
C02652=1046.259,91.631,-85.383,170.441,35.938,156.762
C02653=1046.253,91.382,-85.363,170.439,35.937,156.762
C02654=1046.247,91.133,-85.344,170.437,35.935,156.762
C02655=1046.241,90.884,-85.325,170.436,35.933,156.761
C02656=1046.234,90.634,-85.306,170.434,35.931,156.761
C02657=1046.229,90.385,-85.287,170.431,35.930,156.761
C02658=1046.222,90.136,-85.268,170.430,35.929,156.761
C02659=1046.217,89.887,-85.249,170.428,35.927,156.760
C02660=1046.210,89.637,-85.230,170.426,35.926,156.760
C02661=1046.204,89.388,-85.212,170.425,35.924,156.760
C02662=1046.197,89.139,-85.193,170.423,35.923,156.759
C02663=1046.192,88.890,-85.174,170.421,35.921,156.759
C02664=1046.185,88.641,-85.155,170.419,35.919,156.759
C02665=1046.179,88.391,-85.136,170.417,35.918,156.759
C02666=1046.172,88.142,-85.118,170.415,35.916,156.758
C02667=1046.166,87.892,-85.098,170.414,35.915,156.758
C02668=1046.160,87.643,-85.080,170.412,35.914,156.758
C02669=1046.153,87.394,-85.061,170.410,35.912,156.758
C02670=1046.147,87.145,-85.042,170.409,35.911,156.757
C02671=1046.141,86.895,-85.023,170.406,35.909,156.757
C02672=1046.135,86.646,-85.004,170.404,35.907,156.757
C02673=1046.128,86.397,-84.986,170.403,35.906,156.756
C02674=1046.122,86.148,-84.967,170.401,35.904,156.756
C02675=1046.116,85.900,-84.949,170.399,35.903,156.756
C02676=1046.110,85.650,-84.930,170.398,35.901,156.756
C02677=1046.104,85.401,-84.911,170.396,35.900,156.755
C02678=1046.098,85.152,-84.892,170.393,35.898,156.755
C02679=1046.091,84.903,-84.874,170.392,35.897,156.755
C02680=1046.085,84.653,-84.854,170.390,35.895,156.755
C02681=1046.079,84.404,-84.836,170.389,35.893,156.754
C02682=1046.073,84.155,-84.817,170.387,35.892,156.754
C02683=1046.066,83.905,-84.799,170.385,35.890,156.754
C02684=1046.061,83.656,-84.780,170.384,35.889,156.753
C02685=1046.054,83.407,-84.761,170.382,35.888,156.753
C02686=1046.048,83.158,-84.743,170.379,35.886,156.753
C02687=1046.041,82.909,-84.724,170.378,35.885,156.753
C02688=1046.035,82.659,-84.705,170.376,35.883,156.752
C02689=1046.029,82.410,-84.686,170.374,35.881,156.752
C02690=1046.023,82.160,-84.668,170.373,35.880,156.752
C02691=1046.017,81.911,-84.649,170.371,35.878,156.751
C02692=1046.011,81.663,-84.631,170.368,35.876,156.751
C02693=1046.005,81.414,-84.613,170.367,35.875,156.751
C02694=1045.999,81.164,-84.593,170.365,35.874,156.751
C02695=1045.993,80.914,-84.575,170.363,35.872,156.750
C02696=1045.986,80.665,-84.557,170.362,35.871,156.750
C02697=1045.980,80.416,-84.538,170.360,35.869,156.750
C02698=1045.973,80.167,-84.519,170.359,35.867,156.749
C02699=1045.968,79.917,-84.501,170.357,35.866,156.749
C02700=1045.962,79.669,-84.483,170.354,35.864,156.749
C02701=1045.956,79.420,-84.464,170.353,35.862,156.748
C02702=1045.949,79.170,-84.445,170.351,35.861,156.748
C02703=1045.943,78.921,-84.427,170.349,35.859,156.748
C02704=1045.938,78.671,-84.408,170.348,35.858,156.748
C02705=1045.931,78.422,-84.389,170.346,35.857,156.747
C02706=1045.925,78.173,-84.371,170.344,35.855,156.747
C02707=1045.919,77.924,-84.353,170.342,35.854,156.747
C02708=1045.911,77.638,-84.332,170.340,35.852,156.747
C02709=1045.904,77.352,-84.311,170.338,35.850,156.746
C02710=1045.897,77.066,-84.290,170.336,35.848,156.746
C02711=1045.890,76.780,-84.268,170.334,35.847,156.746
C02712=1045.884,76.531,-84.251,170.333,35.845,156.745
C02713=1045.878,76.282,-84.232,170.331,35.843,156.745
C02714=1045.872,76.032,-84.214,170.328,35.842,156.745
C02715=1045.865,75.783,-84.196,170.327,35.840,156.744
C02716=1045.859,75.534,-84.177,170.325,35.839,156.744
C02717=1045.853,75.284,-84.159,170.323,35.838,156.744
C02718=1045.846,75.035,-84.141,170.322,35.836,156.744
C02719=1045.840,74.786,-84.123,170.320,35.834,156.743
C02720=1045.834,74.537,-84.105,170.318,35.833,156.743
C02721=1045.828,74.287,-84.087,170.316,35.831,156.743
C02722=1045.821,74.038,-84.068,170.314,35.830,156.743
C02723=1045.815,73.788,-84.050,170.312,35.829,156.742
C02724=1045.809,73.540,-84.032,170.311,35.827,156.742
C02725=1045.803,73.290,-84.014,170.309,35.826,156.742
C02726=1045.797,73.041,-83.995,170.307,35.824,156.741
C02727=1045.790,72.792,-83.977,170.306,35.822,156.741
C02728=1045.784,72.542,-83.959,170.304,35.821,156.741
C02729=1045.779,72.293,-83.941,170.302,35.819,156.741
C02730=1045.772,72.044,-83.923,170.300,35.818,156.740
C02731=1045.766,71.794,-83.905,170.298,35.817,156.740
C02732=1045.759,71.546,-83.887,170.297,35.815,156.740
C02733=1045.753,71.296,-83.869,170.295,35.813,156.740
C02734=1045.747,71.047,-83.850,170.293,35.812,156.739
C02735=1045.741,70.798,-83.832,170.292,35.810,156.739
C02736=1045.734,70.549,-83.814,170.290,35.809,156.739
C02737=1045.728,70.299,-83.796,170.287,35.807,156.739
C02738=1045.722,70.050,-83.778,170.286,35.806,156.738
C02739=1045.716,69.801,-83.760,170.284,35.805,156.738
C02740=1045.709,69.551,-83.742,170.282,35.803,156.738
C02741=1045.703,69.302,-83.724,170.281,35.801,156.737
C02742=1045.698,69.053,-83.706,170.279,35.800,156.737
C02743=1045.691,68.803,-83.688,170.277,35.798,156.737
C02744=1045.685,68.554,-83.669,170.275,35.797,156.737
C02745=1045.678,68.305,-83.652,170.273,35.796,156.736
C02746=1045.673,68.056,-83.635,170.272,35.794,156.736
C02747=1045.666,67.807,-83.616,170.270,35.792,156.736
C02748=1045.660,67.557,-83.598,170.268,35.791,156.736
C02749=1045.653,67.307,-83.581,170.267,35.789,156.735
C02750=1045.647,67.059,-83.562,170.265,35.788,156.735
C02751=1045.641,66.809,-83.544,170.263,35.787,156.735
C02752=1045.634,66.560,-83.527,170.261,35.785,156.734
C02753=1045.629,66.311,-83.509,170.259,35.783,156.734
C02754=1045.622,66.062,-83.491,170.257,35.782,156.734
C02755=1045.616,65.812,-83.473,170.256,35.781,156.734
C02756=1045.609,65.563,-83.456,170.254,35.779,156.733
C02757=1045.604,65.314,-83.437,170.252,35.778,156.733
C02758=1045.598,65.064,-83.419,170.251,35.776,156.733
C02759=1045.591,64.815,-83.402,170.249,35.775,156.733
C02760=1045.585,64.566,-83.384,170.246,35.773,156.732
C02761=1045.579,64.316,-83.367,170.245,35.772,156.732
C02762=1045.572,64.067,-83.348,170.243,35.770,156.732
C02763=1045.566,63.818,-83.331,170.241,35.769,156.732
C02764=1045.559,63.569,-83.314,170.240,35.768,156.731
C02765=1045.553,63.319,-83.296,170.238,35.766,156.731
C02766=1045.547,63.070,-83.278,170.236,35.765,156.731
C02767=1045.541,62.821,-83.261,170.235,35.763,156.731
C02768=1045.534,62.571,-83.243,170.232,35.762,156.730
C02769=1045.528,62.322,-83.225,170.230,35.760,156.730
C02770=1045.521,62.073,-83.207,170.229,35.759,156.730
C02771=1045.515,61.824,-83.190,170.227,35.758,156.730
C02772=1045.507,61.537,-83.170,170.225,35.756,156.729
C02773=1045.500,61.251,-83.150,170.223,35.755,156.729
C02774=1045.492,60.965,-83.130,170.221,35.753,156.729
C02775=1045.486,60.679,-83.110,170.219,35.751,156.729
C02776=1045.479,60.429,-83.092,170.217,35.750,156.728
C02777=1045.473,60.180,-83.075,170.215,35.748,156.728
C02778=1045.466,59.931,-83.058,170.213,35.747,156.728
C02779=1045.460,59.681,-83.040,170.211,35.746,156.728
C02780=1045.454,59.432,-83.023,170.210,35.744,156.727
C02781=1045.448,59.183,-83.005,170.208,35.743,156.727
C02782=1045.441,58.933,-82.987,170.206,35.741,156.727
C02783=1045.435,58.685,-82.970,170.205,35.740,156.727
C02784=1045.429,58.435,-82.953,170.203,35.739,156.726
C02785=1045.422,58.185,-82.935,170.200,35.737,156.726
C02786=1045.416,57.936,-82.918,170.199,35.735,156.726
C02787=1045.409,57.687,-82.900,170.197,35.734,156.726
C02788=1045.402,57.437,-82.883,170.195,35.733,156.725
C02789=1045.397,57.188,-82.865,170.194,35.732,156.725
C02790=1045.390,56.939,-82.848,170.192,35.730,156.725
C02791=1045.385,56.690,-82.831,170.190,35.728,156.724
C02792=1045.378,56.441,-82.813,170.189,35.727,156.724
C02793=1045.371,56.191,-82.796,170.187,35.726,156.724
C02794=1045.365,55.942,-82.778,170.184,35.725,156.724
C02795=1045.358,55.693,-82.761,170.183,35.723,156.724
C02796=1045.353,55.444,-82.743,170.181,35.721,156.723
C02797=1045.346,55.194,-82.726,170.179,35.720,156.723
C02798=1045.340,54.945,-82.710,170.178,35.719,156.723
C02799=1045.334,54.695,-82.692,170.176,35.718,156.723
C02800=1045.327,54.446,-82.674,170.174,35.716,156.722
C02801=1045.322,54.197,-82.657,170.173,35.714,156.722
C02802=1045.315,53.947,-82.640,170.170,35.713,156.722
C02803=1045.309,53.698,-82.623,170.168,35.712,156.722
C02804=1045.302,53.449,-82.605,170.167,35.710,156.721
C02805=1045.296,53.200,-82.588,170.165,35.709,156.721
C02806=1045.290,52.950,-82.571,170.163,35.707,156.721
C02807=1045.284,52.701,-82.554,170.162,35.706,156.721
C02808=1045.277,52.451,-82.536,170.160,35.704,156.720
C02809=1045.272,52.202,-82.519,170.158,35.703,156.720
C02810=1045.265,51.953,-82.501,170.156,35.701,156.720
C02811=1045.259,51.704,-82.485,170.154,35.700,156.719
C02812=1045.253,51.454,-82.467,170.152,35.699,156.719
C02813=1045.247,51.205,-82.450,170.151,35.697,156.719
C02814=1045.240,50.956,-82.433,170.149,35.696,156.719
C02815=1045.234,50.707,-82.415,170.147,35.694,156.718
C02816=1045.228,50.457,-82.399,170.146,35.693,156.718
C02817=1045.221,50.208,-82.382,170.144,35.691,156.718
C02818=1045.215,49.958,-82.364,170.142,35.690,156.718
C02819=1045.209,49.709,-82.347,170.140,35.689,156.717
C02820=1045.202,49.459,-82.330,170.138,35.687,156.717
C02821=1045.197,49.210,-82.313,170.136,35.685,156.717
C02822=1045.190,48.961,-82.295,170.135,35.684,156.717
C02823=1045.184,48.712,-82.279,170.133,35.683,156.716
C02824=1045.178,48.462,-82.261,170.131,35.681,156.716
C02825=1045.172,48.213,-82.244,170.130,35.680,156.716
C02826=1045.165,47.963,-82.227,170.128,35.678,156.716
C02827=1045.160,47.714,-82.210,170.126,35.677,156.715
C02828=1045.153,47.465,-82.193,170.123,35.675,156.715
C02829=1045.147,47.215,-82.176,170.122,35.674,156.715
C02830=1045.141,46.966,-82.159,170.120,35.673,156.715
C02831=1045.134,46.717,-82.141,170.118,35.671,156.714
C02832=1045.128,46.467,-82.125,170.117,35.669,156.714
C02833=1045.123,46.218,-82.108,170.115,35.668,156.714
C02834=1045.116,45.969,-82.090,170.113,35.667,156.714
C02835=1045.110,45.720,-82.074,170.112,35.665,156.713
C02836=1045.103,45.446,-82.055,170.109,35.664,156.713
C02837=1045.097,45.173,-82.036,170.107,35.662,156.713
C02838=1045.090,44.900,-82.018,170.105,35.660,156.712
C02839=1045.084,44.627,-81.999,170.103,35.658,156.712
C02840=1045.077,44.377,-81.982,170.102,35.657,156.712
C02841=1045.071,44.129,-81.965,170.100,35.656,156.712
C02842=1045.065,43.879,-81.948,170.098,35.655,156.711
C02843=1045.059,43.630,-81.931,170.097,35.653,156.711
C02844=1045.053,43.380,-81.914,170.094,35.651,156.711
C02845=1045.046,43.132,-81.897,170.092,35.650,156.711
C02846=1045.040,42.882,-81.881,170.091,35.649,156.710
C02847=1045.034,42.633,-81.863,170.089,35.647,156.710
C02848=1045.028,42.382,-81.847,170.087,35.646,156.710
C02849=1045.021,42.134,-81.830,170.086,35.644,156.710
C02850=1045.016,41.884,-81.813,170.084,35.643,156.709
C02851=1045.009,41.635,-81.796,170.082,35.642,156.709
C02852=1045.003,41.386,-81.780,170.081,35.640,156.709
C02853=1044.996,41.136,-81.763,170.078,35.639,156.709
C02854=1044.990,40.887,-81.746,170.076,35.637,156.708
C02855=1044.984,40.637,-81.730,170.074,35.636,156.708
C02856=1044.977,40.374,-81.712,170.073,35.635,156.708
C02857=1044.970,40.112,-81.694,170.071,35.633,156.708
C02858=1044.964,39.849,-81.676,170.069,35.631,156.707
C02859=1044.957,39.586,-81.659,170.067,35.630,156.707
C02860=1044.951,39.338,-81.643,170.066,35.629,156.707
C02861=1044.944,39.088,-81.626,170.064,35.627,156.707
C02862=1044.938,38.838,-81.610,170.061,35.626,156.707
C02863=1044.933,38.589,-81.592,170.059,35.624,156.706
C02864=1044.926,38.339,-81.575,170.058,35.623,156.706
C02865=1044.920,38.090,-81.559,170.056,35.622,156.706
C02866=1044.914,37.841,-81.542,170.054,35.620,156.706
C02867=1044.908,37.591,-81.526,170.053,35.619,156.705
C02868=1044.902,37.342,-81.509,170.051,35.618,156.705
C02869=1044.895,37.093,-81.493,170.049,35.616,156.705
C02870=1044.888,36.843,-81.476,170.048,35.615,156.705
C02871=1044.882,36.594,-81.460,170.045,35.613,156.704
C02872=1044.876,36.344,-81.444,170.043,35.612,156.704
C02873=1044.869,36.095,-81.426,170.041,35.611,156.704
C02874=1044.863,35.846,-81.410,170.040,35.609,156.704
C02875=1044.857,35.597,-81.395,170.038,35.608,156.703
C02876=1044.850,35.347,-81.378,170.036,35.607,156.703
C02877=1044.844,35.098,-81.361,170.034,35.605,156.703
C02878=1044.838,34.849,-81.345,170.033,35.604,156.703
C02879=1044.832,34.599,-81.328,170.031,35.603,156.703
C02880=1044.825,34.349,-81.312,170.029,35.602,156.702
C02881=1044.819,34.100,-81.296,170.027,35.600,156.702
C02882=1044.813,33.851,-81.279,170.025,35.599,156.702
C02883=1044.806,33.601,-81.263,170.023,35.598,156.702
C02884=1044.800,33.352,-81.246,170.021,35.596,156.701
C02885=1044.794,33.103,-81.230,170.020,35.594,156.701
C02886=1044.788,32.853,-81.214,170.018,35.593,156.701
C02887=1044.781,32.604,-81.198,170.016,35.592,156.701
C02888=1044.775,32.355,-81.181,170.014,35.591,156.700
C02889=1044.769,32.105,-81.165,170.013,35.589,156.700
C02890=1044.763,31.856,-81.148,170.011,35.588,156.700
C02891=1044.756,31.606,-81.132,170.008,35.587,156.700
C02892=1044.749,31.357,-81.116,170.007,35.585,156.699
C02893=1044.743,31.108,-81.100,170.005,35.584,156.699
C02894=1044.738,30.858,-81.083,170.003,35.583,156.699
C02895=1044.731,30.608,-81.067,170.001,35.581,156.699
C02896=1044.725,30.359,-81.051,170.000,35.579,156.698
C02897=1044.718,30.110,-81.034,169.998,35.578,156.698
C02898=1044.712,29.861,-81.018,169.996,35.577,156.698
C02899=1044.706,29.612,-81.002,169.994,35.576,156.698
C02900=1044.699,29.325,-80.984,169.992,35.574,156.698
C02901=1044.692,29.038,-80.964,169.989,35.572,156.697
C02902=1044.684,28.751,-80.946,169.987,35.571,156.697
C02903=1044.677,28.465,-80.927,169.985,35.570,156.697
C02904=1044.671,28.216,-80.911,169.984,35.568,156.697
C02905=1044.664,27.967,-80.895,169.982,35.567,156.696
C02906=1044.658,27.717,-80.879,169.980,35.566,156.696
C02907=1044.652,27.467,-80.863,169.978,35.565,156.696
C02908=1044.645,27.218,-80.847,169.977,35.563,156.696
C02909=1044.640,26.968,-80.831,169.975,35.562,156.695
C02910=1044.633,26.719,-80.815,169.972,35.561,156.695
C02911=1044.627,26.470,-80.799,169.970,35.559,156.695
C02912=1044.621,26.221,-80.783,169.969,35.558,156.695
C02913=1044.614,25.971,-80.767,169.967,35.557,156.695
C02914=1044.608,25.722,-80.750,169.965,35.555,156.694
C02915=1044.601,25.473,-80.735,169.963,35.554,156.694
C02916=1044.595,25.223,-80.719,169.962,35.553,156.694
C02917=1044.589,24.974,-80.702,169.960,35.551,156.694
C02918=1044.582,24.724,-80.686,169.958,35.550,156.694
C02919=1044.576,24.474,-80.671,169.956,35.549,156.693
C02920=1044.569,24.225,-80.655,169.955,35.548,156.693
C02921=1044.564,23.976,-80.639,169.952,35.546,156.693
C02922=1044.557,23.727,-80.623,169.950,35.545,156.693
C02923=1044.551,23.477,-80.607,169.948,35.544,156.692
C02924=1044.545,23.228,-80.591,169.947,35.542,156.692
C02925=1044.538,22.978,-80.575,169.945,35.541,156.692
C02926=1044.532,22.728,-80.559,169.943,35.540,156.692
C02927=1044.525,22.479,-80.543,169.941,35.538,156.692
C02928=1044.519,22.230,-80.527,169.939,35.537,156.691
C02929=1044.513,21.981,-80.511,169.938,35.536,156.691
C02930=1044.507,21.731,-80.496,169.936,35.535,156.691
C02931=1044.500,21.482,-80.480,169.933,35.533,156.691
C02932=1044.494,21.233,-80.464,169.931,35.532,156.690
C02933=1044.488,20.983,-80.448,169.930,35.531,156.690
C02934=1044.482,20.734,-80.433,169.928,35.529,156.690
C02935=1044.475,20.483,-80.416,169.926,35.528,156.690
C02936=1044.469,20.234,-80.401,169.924,35.527,156.690
C02937=1044.463,19.985,-80.384,169.923,35.525,156.689
C02938=1044.456,19.735,-80.369,169.921,35.524,156.689
C02939=1044.451,19.486,-80.353,169.919,35.523,156.689
C02940=1044.444,19.237,-80.337,169.917,35.521,156.689
C02941=1044.437,18.987,-80.322,169.915,35.520,156.688
C02942=1044.431,18.738,-80.306,169.913,35.519,156.688
C02943=1044.425,18.489,-80.291,169.911,35.518,156.688
C02944=1044.419,18.239,-80.275,169.909,35.516,156.688
C02945=1044.412,17.990,-80.259,169.907,35.515,156.688
C02946=1044.406,17.741,-80.244,169.905,35.514,156.687
C02947=1044.400,17.490,-80.228,169.904,35.512,156.687
C02948=1044.393,17.241,-80.212,169.902,35.511,156.687
C02949=1044.387,16.992,-80.196,169.900,35.510,156.687
C02950=1044.381,16.742,-80.181,169.898,35.509,156.687
C02951=1044.374,16.493,-80.165,169.897,35.508,156.686
C02952=1044.368,16.243,-80.150,169.895,35.506,156.686
C02953=1044.361,15.994,-80.134,169.892,35.505,156.686
C02954=1044.356,15.745,-80.118,169.890,35.504,156.686
C02955=1044.349,15.495,-80.103,169.888,35.502,156.685
C02956=1044.342,15.246,-80.087,169.887,35.501,156.685
C02957=1044.337,14.996,-80.072,169.885,35.500,156.685
C02958=1044.330,14.747,-80.056,169.883,35.499,156.685
C02959=1044.324,14.497,-80.040,169.881,35.497,156.685
C02960=1044.318,14.248,-80.025,169.879,35.496,156.684
C02961=1044.311,13.998,-80.010,169.878,35.495,156.684
C02962=1044.305,13.749,-79.994,169.876,35.494,156.684
C02963=1044.298,13.500,-79.979,169.874,35.493,156.684
C02964=1044.292,13.214,-79.961,169.871,35.491,156.684
C02965=1044.284,12.929,-79.943,169.869,35.490,156.683
C02966=1044.276,12.644,-79.926,169.867,35.489,156.683
C02967=1044.270,12.359,-79.908,169.865,35.487,156.683
C02968=1044.263,12.110,-79.893,169.863,35.486,156.683
C02969=1044.257,11.860,-79.878,169.861,35.485,156.683
C02970=1044.250,11.611,-79.863,169.859,35.483,156.682
C02971=1044.244,11.361,-79.848,169.857,35.482,156.682
C02972=1044.238,11.112,-79.832,169.855,35.481,156.682
C02973=1044.231,10.862,-79.817,169.854,35.480,156.682
C02974=1044.225,10.613,-79.802,169.852,35.479,156.682
C02975=1044.218,10.364,-79.786,169.850,35.477,156.681
C02976=1044.212,10.114,-79.771,169.847,35.476,156.681
C02977=1044.205,9.865,-79.755,169.845,35.475,156.681
C02978=1044.199,9.615,-79.740,169.843,35.474,156.681
C02979=1044.192,9.366,-79.725,169.842,35.473,156.681
C02980=1044.186,9.116,-79.709,169.840,35.472,156.680
C02981=1044.180,8.867,-79.694,169.838,35.470,156.680
C02982=1044.174,8.617,-79.679,169.836,35.469,156.680
C02983=1044.167,8.368,-79.664,169.834,35.468,156.680
C02984=1044.161,8.118,-79.649,169.832,35.467,156.680
C02985=1044.154,7.869,-79.634,169.831,35.466,156.679
C02986=1044.148,7.619,-79.619,169.829,35.464,156.679
C02987=1044.141,7.370,-79.603,169.827,35.463,156.679
C02988=1044.135,7.120,-79.588,169.824,35.462,156.679
C02989=1044.129,6.870,-79.573,169.822,35.461,156.679
C02990=1044.123,6.621,-79.558,169.820,35.460,156.678
C02991=1044.117,6.372,-79.542,169.818,35.458,156.678
C02992=1044.110,6.123,-79.527,169.817,35.457,156.678
C02993=1044.104,5.873,-79.513,169.815,35.456,156.678
C02994=1044.098,5.623,-79.498,169.813,35.455,156.678
C02995=1044.091,5.374,-79.482,169.811,35.454,156.677
C02996=1044.084,5.125,-79.467,169.809,35.452,156.677
C02997=1044.078,4.875,-79.452,169.807,35.451,156.677
C02998=1044.072,4.626,-79.437,169.806,35.450,156.677
C02999=1044.067,4.376,-79.422,169.804,35.449,156.677
C03000=1044.060,4.127,-79.406,169.801,35.448,156.676
C03001=1044.054,3.877,-79.391,169.799,35.446,156.676
C03002=1044.047,3.628,-79.376,169.797,35.445,156.676
C03003=1044.041,3.378,-79.361,169.795,35.444,156.676
C03004=1044.034,3.128,-79.346,169.793,35.443,156.676
C03005=1044.029,2.879,-79.332,169.792,35.442,156.675
C03006=1044.022,2.630,-79.316,169.790,35.441,156.675
C03007=1044.016,2.381,-79.301,169.788,35.439,156.675
C03008=1044.009,2.131,-79.286,169.786,35.438,156.675
C03009=1044.003,1.881,-79.271,169.784,35.437,156.675
C03010=1043.997,1.632,-79.257,169.782,35.436,156.674
C03011=1043.991,1.383,-79.242,169.780,35.435,156.674
C03012=1043.984,1.133,-79.227,169.779,35.433,156.674
C03013=1043.979,0.883,-79.211,169.776,35.432,156.674
C03014=1043.972,0.633,-79.196,169.774,35.431,156.674
C03015=1043.966,0.385,-79.182,169.772,35.430,156.673
C03016=1043.960,0.135,-79.167,169.770,35.429,156.673
C03017=1043.953,-0.114,-79.151,169.768,35.427,156.673
C03018=1043.947,-0.364,-79.136,169.766,35.426,156.673
C03019=1043.941,-0.613,-79.122,169.765,35.425,156.673
C03020=1043.935,-0.862,-79.107,169.763,35.424,156.673
C03021=1043.928,-1.112,-79.092,169.761,35.423,156.672
C03022=1043.922,-1.362,-79.077,169.759,35.421,156.672
C03023=1043.916,-1.611,-79.062,169.757,35.420,156.672
C03024=1043.910,-1.860,-79.047,169.755,35.419,156.672
C03025=1043.904,-2.110,-79.032,169.752,35.418,156.672
C03026=1043.897,-2.360,-79.017,169.750,35.417,156.671
C03027=1043.891,-2.609,-79.003,169.749,35.415,156.671
C03028=1043.884,-2.892,-78.987,169.746,35.414,156.671
C03029=1043.878,-3.176,-78.970,169.744,35.413,156.671
C03030=1043.871,-3.459,-78.953,169.742,35.411,156.670
C03031=1043.863,-3.742,-78.936,169.740,35.410,156.670
C03032=1043.857,-3.992,-78.921,169.738,35.409,156.670
C03033=1043.851,-4.242,-78.906,169.736,35.408,156.670
C03034=1043.844,-4.491,-78.892,169.734,35.407,156.670
C03035=1043.837,-4.741,-78.877,169.732,35.405,156.670
C03036=1043.832,-4.990,-78.863,169.731,35.405,156.669
C03037=1043.825,-5.239,-78.849,169.729,35.403,156.669
C03038=1043.818,-5.489,-78.834,169.726,35.403,156.669
C03039=1043.812,-5.739,-78.819,169.724,35.401,156.669
C03040=1043.806,-5.988,-78.804,169.722,35.400,156.669
C03041=1043.799,-6.237,-78.790,169.720,35.399,156.669
C03042=1043.793,-6.487,-78.776,169.718,35.398,156.668
C03043=1043.787,-6.736,-78.761,169.716,35.397,156.668
C03044=1043.781,-6.986,-78.746,169.714,35.396,156.668
C03045=1043.774,-7.235,-78.732,169.712,35.395,156.668
C03046=1043.768,-7.486,-78.718,169.710,35.394,156.668
C03047=1043.762,-7.735,-78.703,169.708,35.393,156.667
C03048=1043.755,-7.984,-78.689,169.706,35.391,156.667
C03049=1043.748,-8.234,-78.674,169.705,35.391,156.667
C03050=1043.743,-8.483,-78.660,169.703,35.389,156.667
C03051=1043.736,-8.732,-78.645,169.701,35.389,156.667
C03052=1043.729,-8.982,-78.631,169.699,35.387,156.667
C03053=1043.723,-9.231,-78.616,169.696,35.386,156.666
C03054=1043.717,-9.481,-78.602,169.694,35.385,156.666
C03055=1043.710,-9.731,-78.587,169.692,35.384,156.666
C03056=1043.704,-9.980,-78.573,169.690,35.383,156.666
C03057=1043.698,-10.230,-78.559,169.688,35.382,156.666
C03058=1043.691,-10.479,-78.544,169.686,35.381,156.666
C03059=1043.685,-10.728,-78.530,169.684,35.380,156.665
C03060=1043.679,-10.978,-78.515,169.682,35.379,156.665
C03061=1043.673,-11.227,-78.501,169.680,35.377,156.665
C03062=1043.667,-11.477,-78.486,169.678,35.377,156.665
C03063=1043.660,-11.727,-78.472,169.676,35.375,156.665
C03064=1043.654,-11.976,-78.458,169.675,35.375,156.665
C03065=1043.648,-12.225,-78.443,169.673,35.373,156.664
C03066=1043.642,-12.475,-78.429,169.671,35.372,156.664
C03067=1043.635,-12.724,-78.415,169.669,35.371,156.664
C03068=1043.629,-12.975,-78.401,169.666,35.370,156.664
C03069=1043.623,-13.224,-78.386,169.664,35.369,156.664
C03070=1043.616,-13.473,-78.372,169.662,35.368,156.664
C03071=1043.610,-13.722,-78.358,169.660,35.367,156.663
C03072=1043.604,-13.972,-78.343,169.658,35.366,156.663
C03073=1043.598,-14.221,-78.330,169.656,35.365,156.663
C03074=1043.591,-14.471,-78.315,169.654,35.363,156.663
C03075=1043.585,-14.721,-78.301,169.652,35.363,156.663
C03076=1043.579,-14.970,-78.287,169.650,35.361,156.663
C03077=1043.573,-15.220,-78.272,169.648,35.360,156.662
C03078=1043.567,-15.469,-78.258,169.646,35.359,156.662
C03079=1043.560,-15.719,-78.244,169.644,35.358,156.662
C03080=1043.554,-15.968,-78.230,169.642,35.357,156.662
C03081=1043.548,-16.218,-78.216,169.640,35.356,156.662
C03082=1043.541,-16.467,-78.202,169.638,35.355,156.662
C03083=1043.535,-16.717,-78.188,169.635,35.354,156.661
C03084=1043.528,-16.966,-78.173,169.633,35.353,156.661
C03085=1043.522,-17.216,-78.160,169.631,35.352,156.661
C03086=1043.516,-17.466,-78.146,169.629,35.351,156.661
C03087=1043.509,-17.715,-78.132,169.627,35.350,156.661
C03088=1043.503,-17.965,-78.118,169.625,35.349,156.661
C03089=1043.496,-18.213,-78.104,169.623,35.348,156.661
C03090=1043.490,-18.464,-78.090,169.621,35.348,156.660
C03091=1043.484,-18.714,-78.076,169.619,35.346,156.660
C03092=1043.477,-18.995,-78.060,169.617,35.345,156.660
C03093=1043.469,-19.277,-78.044,169.615,35.344,156.660
C03094=1043.463,-19.558,-78.029,169.613,35.343,156.660
C03095=1043.455,-19.840,-78.013,169.610,35.342,156.660
C03096=1043.450,-20.090,-77.999,169.608,35.341,156.659
C03097=1043.442,-20.339,-77.985,169.606,35.340,156.659
C03098=1043.436,-20.588,-77.971,169.604,35.339,156.659
C03099=1043.430,-20.839,-77.957,169.602,35.338,156.659
C03100=1043.424,-21.087,-77.943,169.599,35.337,156.659
C03101=1043.418,-21.338,-77.929,169.597,35.336,156.659
C03102=1043.411,-21.587,-77.916,169.595,35.335,156.658
C03103=1043.405,-21.837,-77.902,169.593,35.334,156.658
C03104=1043.399,-22.086,-77.888,169.591,35.333,156.658
C03105=1043.392,-22.336,-77.874,169.589,35.332,156.658
C03106=1043.386,-22.585,-77.860,169.587,35.331,156.658
C03107=1043.380,-22.835,-77.846,169.585,35.330,156.658
C03108=1043.373,-23.084,-77.832,169.583,35.329,156.658
C03109=1043.368,-23.333,-77.819,169.581,35.328,156.657
C03110=1043.361,-23.583,-77.805,169.579,35.327,156.657
C03111=1043.355,-23.833,-77.792,169.577,35.326,156.657
C03112=1043.348,-24.082,-77.777,169.575,35.325,156.657
C03113=1043.342,-24.332,-77.763,169.573,35.324,156.657
C03114=1043.337,-24.581,-77.750,169.571,35.323,156.657
C03115=1043.330,-24.831,-77.736,169.569,35.323,156.657
C03116=1043.323,-25.080,-77.723,169.567,35.321,156.656
C03117=1043.317,-25.331,-77.708,169.564,35.320,156.656
C03118=1043.311,-25.579,-77.694,169.562,35.319,156.656
C03119=1043.305,-25.829,-77.681,169.560,35.318,156.656
C03120=1043.299,-26.079,-77.667,169.558,35.317,156.656
C03121=1043.292,-26.328,-77.654,169.556,35.316,156.656
C03122=1043.286,-26.577,-77.640,169.554,35.316,156.656
C03123=1043.280,-26.828,-77.626,169.552,35.314,156.655
C03124=1043.274,-27.077,-77.613,169.550,35.314,156.655
C03125=1043.267,-27.327,-77.599,169.548,35.312,156.655
C03126=1043.261,-27.576,-77.586,169.546,35.312,156.655
C03127=1043.255,-27.825,-77.573,169.544,35.311,156.655
C03128=1043.248,-28.075,-77.558,169.542,35.310,156.655
C03129=1043.242,-28.324,-77.544,169.540,35.309,156.654
C03130=1043.235,-28.574,-77.531,169.538,35.308,156.654
C03131=1043.229,-28.824,-77.518,169.536,35.308,156.654
C03132=1043.223,-29.073,-77.504,169.534,35.307,156.654
C03133=1043.216,-29.323,-77.491,169.532,35.305,156.654
C03134=1043.210,-29.572,-77.477,169.530,35.305,156.654
C03135=1043.204,-29.821,-77.464,169.528,35.304,156.654
C03136=1043.197,-30.071,-77.451,169.524,35.303,156.654
C03137=1043.192,-30.322,-77.437,169.522,35.302,156.653
C03138=1043.185,-30.571,-77.424,169.520,35.301,156.653
C03139=1043.179,-30.821,-77.410,169.518,35.301,156.653
C03140=1043.172,-31.070,-77.397,169.516,35.299,156.653
C03141=1043.166,-31.319,-77.384,169.514,35.299,156.653
C03142=1043.159,-31.569,-77.370,169.512,35.298,156.653
C03143=1043.153,-31.818,-77.357,169.510,35.297,156.653
C03144=1043.147,-32.068,-77.344,169.508,35.296,156.653
C03145=1043.140,-32.318,-77.330,169.506,35.295,156.652
C03146=1043.134,-32.567,-77.317,169.504,35.294,156.652
C03147=1043.128,-32.817,-77.303,169.502,35.294,156.652
C03148=1043.122,-33.067,-77.289,169.500,35.292,156.652
C03149=1043.116,-33.316,-77.277,169.498,35.292,156.652
C03150=1043.109,-33.566,-77.264,169.495,35.291,156.652
C03151=1043.103,-33.815,-77.250,169.493,35.290,156.652
C03152=1043.096,-34.065,-77.237,169.491,35.289,156.652
C03153=1043.090,-34.314,-77.223,169.489,35.288,156.651
C03154=1043.084,-34.563,-77.210,169.487,35.287,156.651
C03155=1043.078,-34.813,-77.198,169.485,35.287,156.651
C03156=1043.071,-35.094,-77.182,169.483,35.285,156.651
C03157=1043.063,-35.375,-77.167,169.480,35.285,156.651
C03158=1043.057,-35.656,-77.153,169.477,35.283,156.651
C03159=1043.050,-35.937,-77.137,169.475,35.283,156.651
C03160=1043.044,-36.187,-77.124,169.473,35.282,156.651
C03161=1043.038,-36.436,-77.111,169.471,35.281,156.650
C03162=1043.031,-36.686,-77.097,169.468,35.280,156.650
C03163=1043.025,-36.935,-77.084,169.466,35.279,156.650
C03164=1043.019,-37.185,-77.072,169.464,35.278,156.650
C03165=1043.012,-37.435,-77.058,169.462,35.278,156.650
C03166=1043.006,-37.684,-77.045,169.460,35.276,156.650
C03167=1043.000,-37.933,-77.032,169.458,35.276,156.650
C03168=1042.994,-38.184,-77.019,169.456,35.275,156.650
C03169=1042.987,-38.433,-77.006,169.454,35.274,156.649
C03170=1042.981,-38.682,-76.992,169.452,35.273,156.649
C03171=1042.975,-38.932,-76.980,169.450,35.272,156.649
C03172=1042.969,-39.181,-76.966,169.447,35.272,156.649
C03173=1042.962,-39.431,-76.953,169.445,35.271,156.649
C03174=1042.956,-39.681,-76.940,169.443,35.270,156.649
C03175=1042.949,-39.930,-76.928,169.441,35.269,156.649
C03176=1042.943,-40.180,-76.915,169.439,35.269,156.649
C03177=1042.937,-40.429,-76.902,169.437,35.268,156.649
C03178=1042.930,-40.679,-76.888,169.435,35.267,156.648
C03179=1042.924,-40.929,-76.876,169.433,35.267,156.648
C03180=1042.918,-41.178,-76.863,169.430,35.266,156.648
C03181=1042.912,-41.428,-76.850,169.428,35.265,156.648
C03182=1042.905,-41.677,-76.837,169.425,35.264,156.648
C03183=1042.900,-41.927,-76.825,169.423,35.263,156.648
C03184=1042.893,-42.177,-76.811,169.421,35.262,156.648
C03185=1042.886,-42.426,-76.798,169.419,35.262,156.648
C03186=1042.880,-42.676,-76.786,169.417,35.261,156.648
C03187=1042.874,-42.925,-76.772,169.414,35.260,156.647
C03188=1042.868,-43.175,-76.760,169.412,35.260,156.647
C03189=1042.861,-43.424,-76.747,169.410,35.259,156.647
C03190=1042.855,-43.674,-76.735,169.408,35.258,156.647
C03191=1042.849,-43.923,-76.721,169.406,35.257,156.647
C03192=1042.842,-44.174,-76.708,169.404,35.257,156.647
C03193=1042.836,-44.423,-76.695,169.402,35.256,156.647
C03194=1042.829,-44.673,-76.683,169.399,35.255,156.647
C03195=1042.823,-44.922,-76.671,169.397,35.255,156.647
C03196=1042.817,-45.172,-76.657,169.395,35.254,156.647
C03197=1042.811,-45.422,-76.645,169.393,35.253,156.647
C03198=1042.805,-45.671,-76.632,169.391,35.253,156.646
C03199=1042.798,-45.920,-76.620,169.389,35.252,156.646
C03200=1042.792,-46.170,-76.606,169.386,35.251,156.646
C03201=1042.786,-46.420,-76.594,169.384,35.250,156.646
C03202=1042.780,-46.669,-76.581,169.382,35.250,156.646
C03203=1042.773,-46.918,-76.569,169.380,35.249,156.646
C03204=1042.767,-47.168,-76.556,169.378,35.248,156.646
C03205=1042.761,-47.418,-76.543,169.376,35.248,156.646
C03206=1042.755,-47.667,-76.530,169.374,35.247,156.646
C03207=1042.749,-47.917,-76.518,169.371,35.246,156.646
C03208=1042.742,-48.166,-76.505,169.369,35.245,156.645
C03209=1042.736,-48.417,-76.492,169.367,35.245,156.645
C03210=1042.730,-48.667,-76.479,169.364,35.243,156.645
C03211=1042.723,-48.916,-76.467,169.362,35.243,156.645
C03212=1042.717,-49.166,-76.454,169.360,35.242,156.645
C03213=1042.712,-49.415,-76.442,169.357,35.241,156.645
C03214=1042.706,-49.664,-76.429,169.355,35.240,156.645
C03215=1042.699,-49.914,-76.417,169.353,35.240,156.645
C03216=1042.693,-50.164,-76.404,169.351,35.239,156.645
C03217=1042.687,-50.413,-76.392,169.349,35.238,156.644
C03218=1042.680,-50.663,-76.379,169.346,35.238,156.645
C03219=1042.674,-50.913,-76.366,169.344,35.238,156.644
C03220=1042.667,-51.194,-76.353,169.342,35.237,156.644
C03221=1042.659,-51.475,-76.339,169.339,35.236,156.644
C03222=1042.652,-51.757,-76.324,169.337,35.235,156.644
C03223=1042.645,-52.038,-76.311,169.334,35.235,156.644
C03224=1042.639,-52.288,-76.299,169.332,35.235,156.644
C03225=1042.633,-52.538,-76.287,169.330,35.234,156.644
C03226=1042.625,-52.787,-76.274,169.328,35.233,156.644
C03227=1042.619,-53.037,-76.262,169.325,35.232,156.644
C03228=1042.613,-53.286,-76.249,169.323,35.232,156.644
C03229=1042.607,-53.536,-76.237,169.321,35.232,156.644
C03230=1042.601,-53.785,-76.225,169.319,35.231,156.644
C03231=1042.594,-54.035,-76.213,169.316,35.230,156.644
C03232=1042.588,-54.285,-76.201,169.314,35.230,156.644
C03233=1042.582,-54.534,-76.188,169.312,35.229,156.643
C03234=1042.575,-54.784,-76.176,169.310,35.229,156.643
C03235=1042.569,-55.034,-76.164,169.308,35.228,156.643
C03236=1042.562,-55.283,-76.151,169.305,35.228,156.643
C03237=1042.555,-55.532,-76.139,169.303,35.227,156.643
C03238=1042.550,-55.782,-76.127,169.301,35.226,156.643
C03239=1042.543,-56.032,-76.115,169.299,35.226,156.643
C03240=1042.536,-56.281,-76.103,169.296,35.226,156.643
C03241=1042.530,-56.531,-76.090,169.294,35.225,156.643
C03242=1042.524,-56.781,-76.078,169.292,35.224,156.643
C03243=1042.517,-57.031,-76.066,169.290,35.224,156.643
C03244=1042.511,-57.280,-76.054,169.287,35.223,156.643
C03245=1042.504,-57.530,-76.042,169.285,35.223,156.643
C03246=1042.499,-57.779,-76.030,169.283,35.222,156.643
C03247=1042.493,-58.029,-76.018,169.281,35.222,156.643
C03248=1042.486,-58.278,-76.006,169.278,35.221,156.642
C03249=1042.480,-58.529,-75.994,169.276,35.220,156.642
C03250=1042.474,-58.778,-75.982,169.274,35.220,156.642
C03251=1042.467,-59.028,-75.970,169.272,35.220,156.642
C03252=1042.461,-59.278,-75.957,169.269,35.219,156.642
C03253=1042.454,-59.527,-75.945,169.266,35.218,156.642
C03254=1042.448,-59.776,-75.934,169.264,35.218,156.642
C03255=1042.442,-60.026,-75.921,169.262,35.217,156.642
C03256=1042.436,-60.276,-75.909,169.260,35.217,156.642
C03257=1042.429,-60.525,-75.897,169.257,35.217,156.642
C03258=1042.423,-60.775,-75.885,169.255,35.216,156.642
C03259=1042.417,-61.025,-75.873,169.253,35.215,156.642
C03260=1042.411,-61.274,-75.862,169.251,35.215,156.642
C03261=1042.405,-61.524,-75.849,169.248,35.214,156.642
C03262=1042.398,-61.774,-75.838,169.246,35.214,156.642
C03263=1042.392,-62.023,-75.826,169.244,35.213,156.641
C03264=1042.386,-62.273,-75.813,169.241,35.213,156.642
C03265=1042.380,-62.522,-75.801,169.239,35.212,156.641
C03266=1042.373,-62.772,-75.790,169.237,35.212,156.641
C03267=1042.367,-63.022,-75.778,169.235,35.211,156.641
C03268=1042.361,-63.272,-75.766,169.232,35.211,156.641
C03269=1042.355,-63.521,-75.754,169.230,35.210,156.641
C03270=1042.348,-63.770,-75.742,169.228,35.210,156.641
C03271=1042.343,-64.021,-75.730,169.226,35.209,156.641
C03272=1042.336,-64.270,-75.718,169.223,35.208,156.641
C03273=1042.330,-64.519,-75.707,169.221,35.208,156.641
C03274=1042.324,-64.769,-75.694,169.219,35.208,156.641
C03275=1042.318,-65.019,-75.683,169.217,35.207,156.641
C03276=1042.311,-65.269,-75.671,169.214,35.207,156.641
C03277=1042.305,-65.518,-75.659,169.212,35.206,156.641
C03278=1042.299,-65.768,-75.648,169.210,35.205,156.641
C03279=1042.293,-66.018,-75.636,169.207,35.205,156.641
C03280=1042.287,-66.267,-75.624,169.205,35.205,156.641
C03281=1042.281,-66.516,-75.611,169.203,35.205,156.641
C03282=1042.274,-66.767,-75.600,169.201,35.204,156.640
C03283=1042.268,-67.016,-75.588,169.198,35.203,156.640
C03284=1042.261,-67.299,-75.575,169.196,35.203,156.640
C03285=1042.254,-67.582,-75.562,169.193,35.202,156.640
C03286=1042.247,-67.864,-75.548,169.191,35.202,156.640
C03287=1042.240,-68.147,-75.535,169.188,35.201,156.640
C03288=1042.234,-68.396,-75.524,169.186,35.201,156.640
C03289=1042.228,-68.646,-75.512,169.184,35.200,156.640
C03290=1042.222,-68.895,-75.500,169.181,35.200,156.640
C03291=1042.216,-69.145,-75.489,169.179,35.199,156.640
C03292=1042.209,-69.395,-75.477,169.177,35.199,156.640
C03293=1042.204,-69.644,-75.465,169.174,35.198,156.640
C03294=1042.198,-69.894,-75.453,169.172,35.198,156.640
C03295=1042.191,-70.144,-75.442,169.170,35.198,156.640
C03296=1042.185,-70.393,-75.431,169.168,35.197,156.640
C03297=1042.179,-70.643,-75.418,169.165,35.196,156.640
C03298=1042.173,-70.893,-75.407,169.163,35.196,156.640
C03299=1042.167,-71.142,-75.395,169.161,35.195,156.640
C03300=1042.161,-71.393,-75.384,169.158,35.195,156.640
C03301=1042.155,-71.642,-75.372,169.156,35.195,156.640
C03302=1042.149,-71.892,-75.361,169.154,35.195,156.640
C03303=1042.143,-72.141,-75.349,169.152,35.194,156.639
C03304=1042.136,-72.391,-75.338,169.149,35.193,156.639
C03305=1042.131,-72.640,-75.326,169.147,35.193,156.639
C03306=1042.125,-72.890,-75.314,169.145,35.192,156.639
C03307=1042.118,-73.140,-75.302,169.142,35.192,156.639
C03308=1042.112,-73.389,-75.291,169.140,35.191,156.639
C03309=1042.106,-73.639,-75.280,169.138,35.191,156.639
C03310=1042.101,-73.889,-75.268,169.135,35.191,156.639
C03311=1042.094,-74.138,-75.256,169.133,35.191,156.639
C03312=1042.088,-74.388,-75.245,169.131,35.190,156.639
C03313=1042.082,-74.638,-75.234,169.128,35.190,156.639
C03314=1042.075,-74.888,-75.222,169.126,35.189,156.639
C03315=1042.070,-75.137,-75.211,169.124,35.189,156.639
C03316=1042.063,-75.387,-75.200,169.121,35.189,156.639
C03317=1042.057,-75.636,-75.188,169.119,35.188,156.639
C03318=1042.051,-75.886,-75.177,169.117,35.188,156.639
C03319=1042.044,-76.136,-75.167,169.114,35.188,156.639
C03320=1042.038,-76.385,-75.155,169.112,35.187,156.639
C03321=1042.031,-76.635,-75.144,169.110,35.187,156.639
C03322=1042.026,-76.885,-75.133,169.107,35.187,156.639
C03323=1042.019,-77.134,-75.121,169.105,35.186,156.639
C03324=1042.013,-77.384,-75.110,169.103,35.186,156.639
C03325=1042.007,-77.634,-75.099,169.100,35.186,156.639
C03326=1042.001,-77.884,-75.088,169.098,35.185,156.639
C03327=1041.995,-78.133,-75.076,169.096,35.185,156.639
C03328=1041.989,-78.383,-75.065,169.093,35.185,156.639
C03329=1041.983,-78.633,-75.054,169.091,35.185,156.639
C03330=1041.977,-78.882,-75.043,169.089,35.185,156.639
C03331=1041.970,-79.132,-75.031,169.086,35.184,156.639
C03332=1041.964,-79.381,-75.020,169.084,35.184,156.639
C03333=1041.958,-79.632,-75.009,169.082,35.184,156.639
C03334=1041.952,-79.881,-74.998,169.079,35.184,156.639
C03335=1041.945,-80.131,-74.987,169.077,35.183,156.639
C03336=1041.940,-80.380,-74.976,169.075,35.183,156.639
C03337=1041.933,-80.630,-74.964,169.072,35.183,156.639
C03338=1041.926,-80.879,-74.954,169.070,35.183,156.639
C03339=1041.920,-81.129,-74.943,169.067,35.182,156.639
C03340=1041.914,-81.379,-74.932,169.065,35.182,156.639
C03341=1041.908,-81.629,-74.921,169.063,35.182,156.639
C03342=1041.902,-81.878,-74.910,169.060,35.182,156.639
C03343=1041.895,-82.128,-74.899,169.058,35.181,156.639
C03344=1041.889,-82.378,-74.888,169.055,35.181,156.639
C03345=1041.882,-82.628,-74.878,169.053,35.181,156.639
C03346=1041.877,-82.877,-74.867,169.051,35.181,156.639
C03347=1041.871,-83.127,-74.856,169.048,35.181,156.639
C03348=1041.863,-83.411,-74.843,169.046,35.180,156.639
C03349=1041.856,-83.697,-74.831,169.043,35.180,156.639
C03350=1041.849,-83.981,-74.819,169.040,35.180,156.639
C03351=1041.842,-84.266,-74.806,169.037,35.180,156.639
C03352=1041.836,-84.516,-74.795,169.035,35.180,156.639
C03353=1041.829,-84.766,-74.784,169.033,35.180,156.639
C03354=1041.823,-85.015,-74.773,169.030,35.180,156.639
C03355=1041.817,-85.265,-74.762,169.028,35.180,156.639
C03356=1041.810,-85.514,-74.752,169.025,35.180,156.639
C03357=1041.804,-85.764,-74.741,169.023,35.179,156.639
C03358=1041.798,-86.014,-74.730,169.021,35.179,156.639
C03359=1041.792,-86.264,-74.720,169.018,35.179,156.639
C03360=1041.786,-86.513,-74.709,169.016,35.179,156.639
C03361=1041.780,-86.764,-74.698,169.013,35.179,156.639
C03362=1041.773,-87.013,-74.688,169.011,35.179,156.639
C03363=1041.768,-87.262,-74.677,169.009,35.178,156.639
C03364=1041.761,-87.512,-74.665,169.006,35.178,156.639
C03365=1041.755,-87.762,-74.655,169.004,35.178,156.639
C03366=1041.749,-88.011,-74.644,169.001,35.178,156.639
C03367=1041.742,-88.261,-74.634,168.999,35.178,156.639
C03368=1041.736,-88.510,-74.623,168.997,35.178,156.639
C03369=1041.731,-88.761,-74.613,168.994,35.178,156.639
C03370=1041.724,-89.010,-74.602,168.992,35.178,156.639
C03371=1041.718,-89.260,-74.591,168.989,35.178,156.639
C03372=1041.712,-89.509,-74.580,168.987,35.177,156.639
C03373=1041.705,-89.759,-74.570,168.985,35.177,156.639
C03374=1041.699,-90.009,-74.559,168.982,35.177,156.639
C03375=1041.694,-90.259,-74.549,168.980,35.177,156.639
C03376=1041.687,-90.509,-74.538,168.977,35.177,156.639
C03377=1041.681,-90.758,-74.527,168.975,35.177,156.639
C03378=1041.675,-91.007,-74.517,168.972,35.177,156.639
C03379=1041.669,-91.257,-74.506,168.970,35.176,156.639
C03380=1041.663,-91.508,-74.495,168.968,35.176,156.639
C03381=1041.656,-91.757,-74.485,168.965,35.176,156.639
C03382=1041.651,-92.006,-74.474,168.963,35.176,156.639
C03383=1041.644,-92.256,-74.464,168.960,35.176,156.639
C03384=1041.638,-92.506,-74.453,168.958,35.176,156.639
C03385=1041.632,-92.756,-74.442,168.956,35.176,156.639
C03386=1041.626,-93.005,-74.432,168.953,35.176,156.639
C03387=1041.620,-93.255,-74.421,168.951,35.176,156.639
C03388=1041.613,-93.505,-74.411,168.948,35.176,156.639
C03389=1041.608,-93.755,-74.400,168.946,35.176,156.639
C03390=1041.602,-94.004,-74.390,168.943,35.176,156.639
C03391=1041.596,-94.254,-74.380,168.941,35.175,156.639
C03392=1041.590,-94.503,-74.369,168.939,35.175,156.639
C03393=1041.583,-94.753,-74.359,168.936,35.175,156.639
C03394=1041.578,-95.003,-74.348,168.934,35.175,156.639
C03395=1041.572,-95.253,-74.337,168.931,35.175,156.639
C03396=1041.565,-95.502,-74.327,168.929,35.175,156.639
C03397=1041.560,-95.752,-74.317,168.927,35.175,156.639
C03398=1041.553,-96.001,-74.307,168.924,35.175,156.640
C03399=1041.547,-96.252,-74.296,168.922,35.175,156.640
C03400=1041.541,-96.501,-74.286,168.919,35.175,156.640
C03401=1041.535,-96.751,-74.275,168.917,35.175,156.640
C03402=1041.530,-97.001,-74.265,168.914,35.175,156.640
C03403=1041.523,-97.250,-74.255,168.912,35.175,156.640
C03404=1041.518,-97.500,-74.244,168.910,35.175,156.640
C03405=1041.511,-97.749,-74.234,168.907,35.175,156.640
C03406=1041.505,-98.000,-74.224,168.905,35.175,156.640
C03407=1041.499,-98.249,-74.213,168.902,35.175,156.640
C03408=1041.493,-98.499,-74.204,168.900,35.175,156.640
C03409=1041.486,-98.748,-74.194,168.897,35.175,156.640
C03410=1041.481,-98.998,-74.183,168.895,35.175,156.640
C03411=1041.474,-99.248,-74.173,168.893,35.176,156.640
C03412=1041.467,-99.535,-74.162,168.890,35.176,156.640
C03413=1041.460,-99.822,-74.149,168.888,35.175,156.640
C03414=1041.453,-100.109,-74.138,168.885,35.175,156.640
C03415=1041.446,-100.397,-74.127,168.882,35.176,156.640
C03416=1041.440,-100.646,-74.116,168.879,35.176,156.640
C03417=1041.434,-100.896,-74.106,168.877,35.176,156.640
C03418=1041.427,-101.146,-74.097,168.875,35.176,156.640
C03419=1041.422,-101.395,-74.086,168.872,35.176,156.640
C03420=1041.416,-101.645,-74.076,168.870,35.176,156.640
C03421=1041.408,-101.895,-74.066,168.867,35.176,156.640
C03422=1041.403,-102.145,-74.056,168.865,35.177,156.641
C03423=1041.397,-102.395,-74.046,168.862,35.176,156.641
C03424=1041.390,-102.644,-74.036,168.860,35.176,156.641
C03425=1041.384,-102.894,-74.026,168.857,35.177,156.641
C03426=1041.379,-103.144,-74.016,168.855,35.177,156.641
C03427=1041.372,-103.393,-74.006,168.852,35.177,156.641
C03428=1041.366,-103.643,-73.996,168.850,35.177,156.641
C03429=1041.361,-103.893,-73.986,168.847,35.177,156.641
C03430=1041.354,-104.142,-73.976,168.845,35.177,156.641
C03431=1041.348,-104.392,-73.966,168.842,35.178,156.641
C03432=1041.342,-104.642,-73.957,168.840,35.178,156.641
C03433=1041.336,-104.891,-73.946,168.837,35.178,156.641
C03434=1041.330,-105.141,-73.936,168.835,35.178,156.641
C03435=1041.324,-105.391,-73.927,168.832,35.178,156.641
C03436=1041.318,-105.641,-73.917,168.830,35.178,156.641
C03437=1041.312,-105.890,-73.906,168.828,35.179,156.641
C03438=1041.306,-106.140,-73.897,168.825,35.178,156.641
C03439=1041.300,-106.390,-73.887,168.823,35.178,156.642
C03440=1041.293,-106.639,-73.877,168.820,35.179,156.642
C03441=1041.287,-106.889,-73.868,168.818,35.179,156.642
C03442=1041.281,-107.139,-73.857,168.815,35.179,156.642
C03443=1041.275,-107.388,-73.847,168.813,35.179,156.642
C03444=1041.269,-107.638,-73.838,168.810,35.180,156.642
C03445=1041.263,-107.888,-73.828,168.808,35.180,156.642
C03446=1041.257,-108.138,-73.819,168.805,35.180,156.642
C03447=1041.251,-108.388,-73.809,168.804,35.180,156.642
C03448=1041.244,-108.637,-73.799,168.801,35.180,156.642
C03449=1041.238,-108.887,-73.789,168.799,35.181,156.642
C03450=1041.232,-109.137,-73.779,168.796,35.181,156.642
C03451=1041.226,-109.387,-73.770,168.794,35.181,156.642
C03452=1041.220,-109.636,-73.760,168.791,35.182,156.643
C03453=1041.214,-109.886,-73.750,168.789,35.182,156.643
C03454=1041.208,-110.136,-73.741,168.786,35.182,156.643
C03455=1041.202,-110.386,-73.731,168.784,35.182,156.643
C03456=1041.195,-110.636,-73.722,168.781,35.183,156.643
C03457=1041.189,-110.885,-73.712,168.779,35.183,156.643
C03458=1041.183,-111.135,-73.703,168.776,35.183,156.643
C03459=1041.177,-111.385,-73.693,168.773,35.183,156.643
C03460=1041.171,-111.634,-73.684,168.771,35.184,156.643
C03461=1041.165,-111.884,-73.674,168.768,35.184,156.643
C03462=1041.159,-112.133,-73.664,168.766,35.184,156.643
C03463=1041.153,-112.383,-73.654,168.763,35.184,156.643
C03464=1041.146,-112.633,-73.645,168.761,35.185,156.643
C03465=1041.141,-112.883,-73.635,168.758,35.185,156.644
C03466=1041.135,-113.133,-73.626,168.756,35.185,156.644
C03467=1041.129,-113.383,-73.616,168.753,35.186,156.644
C03468=1041.123,-113.633,-73.607,168.751,35.186,156.644
C03469=1041.117,-113.882,-73.597,168.748,35.186,156.644
C03470=1041.111,-114.132,-73.588,168.746,35.186,156.644
C03471=1041.105,-114.381,-73.578,168.743,35.187,156.644
C03472=1041.099,-114.631,-73.569,168.741,35.187,156.644
C03473=1041.092,-114.881,-73.559,168.738,35.187,156.644
C03474=1041.086,-115.131,-73.550,168.737,35.188,156.644
C03475=1041.080,-115.381,-73.540,168.734,35.188,156.644
C03476=1041.073,-115.666,-73.530,168.731,35.189,156.645
C03477=1041.067,-115.953,-73.519,168.728,35.189,156.645
C03478=1041.059,-116.238,-73.508,168.725,35.189,156.645
C03479=1041.052,-116.525,-73.497,168.723,35.190,156.645
C03480=1041.046,-116.775,-73.488,168.720,35.190,156.645
C03481=1041.040,-117.025,-73.479,168.718,35.190,156.645
C03482=1041.034,-117.274,-73.470,168.715,35.191,156.645
C03483=1041.028,-117.524,-73.460,168.712,35.191,156.645
C03484=1041.022,-117.774,-73.451,168.710,35.191,156.645
C03485=1041.015,-118.023,-73.442,168.707,35.192,156.645
C03486=1041.009,-118.274,-73.433,168.705,35.192,156.646
C03487=1041.004,-118.523,-73.424,168.702,35.193,156.646
C03488=1040.998,-118.773,-73.414,168.700,35.193,156.646
C03489=1040.991,-119.023,-73.405,168.697,35.193,156.646
C03490=1040.985,-119.272,-73.395,168.695,35.194,156.646
C03491=1040.979,-119.523,-73.386,168.692,35.195,156.646
C03492=1040.973,-119.772,-73.377,168.690,35.194,156.646
C03493=1040.967,-120.021,-73.368,168.687,35.195,156.646
C03494=1040.961,-120.272,-73.359,168.684,35.196,156.646
C03495=1040.955,-120.522,-73.349,168.682,35.196,156.647
C03496=1040.949,-120.771,-73.340,168.680,35.197,156.647
C03497=1040.943,-121.021,-73.331,168.678,35.197,156.647
C03498=1040.937,-121.271,-73.322,168.675,35.197,156.647
C03499=1040.930,-121.520,-73.313,168.673,35.198,156.647
C03500=1040.925,-121.770,-73.304,168.670,35.198,156.647
C03501=1040.919,-122.020,-73.295,168.668,35.199,156.647
///RCONF 1,0,0,0,1,0,0,0,0,0,0,0,0,0,0,0,0,0,0,0,0,0,0,0
C03502=1040.913,-122.270,-73.285,168.665,35.199,156.647
C03503=1040.908,-122.519,-73.277,168.663,35.199,156.647
C03504=1040.901,-122.769,-73.268,168.660,35.200,156.648
C03505=1040.894,-123.019,-73.258,168.657,35.200,156.648
C03506=1040.889,-123.269,-73.249,168.655,35.201,156.648
C03507=1040.883,-123.518,-73.240,168.652,35.202,156.648
C03508=1040.877,-123.768,-73.231,168.650,35.202,156.648
C03509=1040.870,-124.018,-73.222,168.647,35.203,156.648
C03510=1040.865,-124.267,-73.213,168.645,35.203,156.648
C03511=1040.859,-124.518,-73.204,168.642,35.203,156.648
C03512=1040.853,-124.767,-73.195,168.640,35.204,156.648
C03513=1040.847,-125.017,-73.187,168.637,35.204,156.649
C03514=1040.840,-125.267,-73.177,168.634,35.205,156.649
C03515=1040.835,-125.517,-73.168,168.632,35.205,156.649
C03516=1040.828,-125.766,-73.160,168.630,35.206,156.649
C03517=1040.822,-126.016,-73.151,168.628,35.207,156.649
C03518=1040.816,-126.266,-73.141,168.625,35.207,156.649
C03519=1040.810,-126.515,-73.134,168.623,35.208,156.649
C03520=1040.804,-126.765,-73.124,168.620,35.208,156.650
C03521=1040.798,-127.016,-73.115,168.617,35.209,156.650
C03522=1040.792,-127.264,-73.107,168.615,35.209,156.650
C03523=1040.786,-127.515,-73.098,168.612,35.210,156.650
C03524=1040.780,-127.764,-73.088,168.610,35.211,156.650
C03525=1040.774,-128.014,-73.079,168.607,35.211,156.650
C03526=1040.770,-128.264,-73.070,168.605,35.210,156.650
C03527=1040.766,-128.514,-73.059,168.603,35.210,156.650
C03528=1040.763,-128.763,-73.049,168.601,35.209,156.650
C03529=1040.761,-129.014,-73.037,168.599,35.208,156.650
C03530=1040.759,-129.263,-73.024,168.597,35.206,156.649
C03531=1040.759,-129.513,-73.012,168.595,35.203,156.649
C03532=1040.759,-129.763,-72.998,168.593,35.200,156.649
C03533=1040.760,-130.014,-72.984,168.591,35.196,156.648
C03534=1040.762,-130.264,-72.970,168.590,35.193,156.647
C03535=1040.765,-130.513,-72.954,168.589,35.188,156.647
C03536=1040.768,-130.764,-72.938,168.587,35.184,156.646
C03537=1040.772,-131.014,-72.922,168.586,35.178,156.645
C03538=1040.778,-131.264,-72.905,168.586,35.173,156.644
C03539=1040.784,-131.514,-72.887,168.584,35.167,156.643
C03540=1040.437,-131.538,-73.145,168.538,35.361,156.676
C03541=1040.431,-131.289,-73.163,168.538,35.368,156.678
C03542=1040.425,-131.039,-73.180,168.539,35.373,156.678
C03543=1040.421,-130.788,-73.196,168.541,35.378,156.679
C03544=1040.418,-130.537,-73.212,168.542,35.383,156.680
C03545=1040.415,-130.288,-73.228,168.543,35.387,156.681
C03546=1040.413,-130.038,-73.242,168.545,35.391,156.682
C03547=1040.413,-129.788,-73.257,168.546,35.395,156.682
C03548=1040.412,-129.537,-73.270,168.548,35.398,156.683
C03549=1040.412,-129.288,-73.283,168.549,35.400,156.683
C03550=1040.414,-129.037,-73.295,168.551,35.402,156.683
C03551=1040.416,-128.788,-73.306,168.553,35.403,156.683
C03552=1040.419,-128.537,-73.317,168.555,35.405,156.684
C03553=1040.423,-128.287,-73.328,168.557,35.405,156.684
C03554=1040.427,-128.038,-73.338,168.560,35.406,156.684
C03555=1040.433,-127.788,-73.347,168.562,35.406,156.684
C03556=1040.439,-127.539,-73.356,168.565,35.405,156.684
C03557=1040.444,-127.289,-73.365,168.567,35.404,156.683
C03558=1040.451,-127.039,-73.374,168.570,35.404,156.683
C03559=1040.457,-126.789,-73.383,168.572,35.403,156.683
C03560=1040.462,-126.540,-73.392,168.575,35.403,156.683
C03561=1040.469,-126.290,-73.400,168.578,35.402,156.683
C03562=1040.475,-126.041,-73.409,168.580,35.401,156.683
C03563=1040.480,-125.790,-73.418,168.583,35.400,156.683
C03564=1040.487,-125.541,-73.427,168.585,35.400,156.682
C03565=1040.493,-125.291,-73.436,168.588,35.399,156.682
C03566=1040.499,-125.041,-73.445,168.591,35.399,156.682
C03567=1040.505,-124.791,-73.453,168.593,35.398,156.682
C03568=1040.511,-124.542,-73.463,168.596,35.397,156.682
C03569=1040.517,-124.292,-73.471,168.598,35.397,156.682
C03570=1040.524,-124.042,-73.480,168.601,35.397,156.682
C03571=1040.530,-123.792,-73.490,168.603,35.396,156.682
C03572=1040.535,-123.543,-73.498,168.605,35.396,156.682
C03573=1040.541,-123.293,-73.508,168.608,35.395,156.681
C03574=1040.547,-123.042,-73.517,168.610,35.395,156.681
C03575=1040.554,-122.794,-73.525,168.613,35.394,156.681
C03576=1040.560,-122.544,-73.535,168.615,35.393,156.681
C03577=1040.566,-122.293,-73.544,168.618,35.393,156.681
C03578=1040.571,-122.044,-73.553,168.620,35.393,156.681
C03579=1040.577,-121.794,-73.563,168.623,35.392,156.681
C03580=1040.584,-121.544,-73.571,168.626,35.392,156.681
C03581=1040.590,-121.295,-73.580,168.628,35.391,156.680
C03582=1040.596,-121.045,-73.590,168.631,35.391,156.680
C03583=1040.602,-120.795,-73.599,168.633,35.390,156.680
C03584=1040.608,-120.545,-73.608,168.636,35.389,156.680
C03585=1040.614,-120.295,-73.618,168.638,35.390,156.680
///RCONF 1,0,0,0,0,0,0,0,0,0,0,0,0,0,0,0,0,0,0,0,0,0,0,0
C03586=1040.620,-120.046,-73.626,168.641,35.389,156.680
C03587=1040.626,-119.796,-73.635,168.643,35.388,156.680
C03588=1040.632,-119.546,-73.645,168.646,35.388,156.680
C03589=1040.638,-119.297,-73.654,168.649,35.387,156.680
C03590=1040.644,-119.047,-73.663,168.651,35.387,156.680
C03591=1040.650,-118.797,-73.672,168.653,35.387,156.679
C03592=1040.656,-118.547,-73.682,168.655,35.386,156.679
C03593=1040.663,-118.298,-73.691,168.658,35.386,156.679
C03594=1040.668,-118.048,-73.699,168.660,35.385,156.679
C03595=1040.674,-117.798,-73.709,168.663,35.385,156.679
C03596=1040.681,-117.549,-73.718,168.666,35.385,156.679
C03597=1040.687,-117.299,-73.728,168.668,35.384,156.679
C03598=1040.693,-117.049,-73.738,168.671,35.383,156.679
C03599=1040.698,-116.799,-73.746,168.673,35.383,156.679
C03600=1040.704,-116.549,-73.756,168.676,35.383,156.678
